//rTrig1(CLK:=xInbound);
//IF rTrig1.Q THEN
//	eState_temp1	:= '';
//	str4debug:='';
//	str4debug	:= CONCAT(STR1:=sInstanceName,STR2:='-');
//	str4debug	:= CONCAT(STR1:=str4debug,STR2:=DINT_TO_STRING(eState));
//	str4debug	:= CONCAT(STR1:=str4debug,STR2:='-');
//	str4debug	:= CONCAT(STR1:=str4debug,STR2:=strState);
//	str4debug	:= CONCAT(STR1:=str4debug,STR2:='-');
//	str4debug	:= CONCAT(STR1:=str4debug,STR2:='inbound');
//	str4debug	:= CONCAT(STR1:=str4debug,STR2:='-');
//	str4debug	:= CONCAT(STR1:=str4debug,STR2:='ON');
//	ADSLOGSTR(msgCtrlMask:=ADSLOG_MSGTYPE_LOG,msgFmtStr:=str4debug,strArg:='');
//END_IF
//fTrig1(CLK:=xInbound);
//IF eState_temp1<>strState THEN
//	eState_temp1	:= strState;
//	state_track	:= CONCAT(STR1:=state_track,STR2:=eState_temp1);
//	state_track	:= CONCAT(STR1:=state_track,STR2:='->');
//END_IF
//IF fTrig1.Q THEN
//	str4debug:='';
//	str4debug	:= CONCAT(STR1:=sInstanceName,STR2:='-');
//	str4debug	:= CONCAT(STR1:=str4debug,STR2:=DINT_TO_STRING(eState));
//	str4debug	:= CONCAT(STR1:=str4debug,STR2:='-');
//	str4debug	:= CONCAT(STR1:=str4debug,STR2:=state_track);
//	str4debug	:= CONCAT(STR1:=str4debug,STR2:='-');
//	str4debug	:= CONCAT(STR1:=str4debug,STR2:='inbound');
//	str4debug	:= CONCAT(STR1:=str4debug,STR2:='-');	
//	str4debug	:= CONCAT(STR1:=str4debug,STR2:='OFF');
//	ADSLOGSTR(msgCtrlMask:=ADSLOG_MSGTYPE_LOG,msgFmtStr:=str4debug,strArg:='');
//END_IF
IF sInstanceName='working1' THEN
	GVL.fb_autoStore1(	eModeCommand:=eModeCommand,
						eMode	=>,
						eState =>stSubModuleInfo[1].eState
					);
	stSubModuleInfo[1].Active			:= FALSE;//while on site,set to FALSE
	IF stSubModuleInfo[1].Active THEN
		eCommand:=eCommand;
	END_IF
	IF  GVL.fb_autoStore1.bUndefinedDone THEN
		bUndefinedDone := TRUE;
	END_IF	
END_IF
IF sInstanceName='working2' THEN
	GVL.fb_autoStore2(	eModeCommand:=eModeCommand,
						eMode	=>,
						eState =>stSubModuleInfo[1].eState
					);
	stSubModuleInfo[1].Active			:= FALSE;//while on site,set to FALSE
	IF stSubModuleInfo[1].Active THEN
		eCommand:=eCommand;
	END_IF	
	IF  GVL.fb_autoStore2.bUndefinedDone THEN
		bUndefinedDone := TRUE;
	END_IF		
END_IF


IF bUndefinedDone AND NOT bMachineStartedUp THEN
	eCommand	:= ePMLCommand_Abort;
	bMachineStartedUp			:= TRUE;
END_IF
//The fbStateMachine from FB_Machine gets the Information about the states and activity from the subunits
fbStateMachine.stSubUnitInfoRef.ArraySize		:= SIZEOF(stSubModuleInfo);
fbStateMachine.stSubUnitInfoRef.NoOfSubUnits	:= iSubModule;
fbStateMachine.stSubUnitInfoRef.pArray			:= ADR(stSubModuleInfo);

(*
Description: 
the callback that will be invoked when there is a publish for what the subscriber was subscribed to.
*)
METHOD Callback
VAR_INPUT
	data : PubSubData;
END_VAR

IF sInstanceName='working1' THEN
	CASE data.Topic OF	
		E_Topics.WORKING1_INBOUND_TOTE:
			IF NOT xInbound AND NOT xOutbound THEN
				xInbound	:= TRUE;
			END_IF
		E_Topics.WORKING1_OUTBOUND_TOTE:
			IF NOT xInbound AND NOT xOutbound THEN
				xOutbound	:= TRUE;
			END_IF
		E_Topics.WORKING1_BEGIN_INBOUND:
			xBeginInbound	:= TRUE;	
		E_Topics.WORKING1_ABORT_INBOUND:
			IF eStates=E_WorkingStates.WAIT_NEW_TOTE THEN
				subData.Topic	:= E_Topics.LOADING_END_OUTBOUND_WOKING1;
				GVL.PubSubService.Publish(topic:=E_Topics.LOADING_END_OUTBOUND_WOKING1,data:= subData);		
				xAbortInbound	:= TRUE;
			END_IF	
		E_Topics.WORKING1_ABORT_OUTBOUND:
			xAbortOutbound	:= TRUE;			

	END_CASE
END_IF
IF sInstanceName='working2' THEN
	CASE data.Topic OF	
		E_Topics.WORKING2_INBOUND_TOTE:
			IF NOT xInbound AND NOT xOutbound THEN
				xInbound	:= TRUE;
			END_IF
		E_Topics.WORKING2_OUTBOUND_TOTE:
			IF NOT xInbound AND NOT xOutbound THEN
				xOutbound	:= TRUE;
			END_IF
		E_Topics.WORKING2_BEGIN_INBOUND:
			xBeginInbound	:= TRUE;	
		E_Topics.WORKING2_ABORT_INBOUND:
			IF eStates=E_WorkingStates.WAIT_NEW_TOTE THEN
				subData.Topic	:= E_Topics.LOADING_END_OUTBOUND_WOKING2;
				GVL.PubSubService.Publish(topic:=E_Topics.LOADING_END_OUTBOUND_WOKING2,data:= subData);				
				xAbortInbound	:= TRUE;
			END_IF
		E_Topics.WORKING2_ABORT_OUTBOUND:
			xAbortOutbound	:= TRUE;	
		
	END_CASE
END_IF
END_METHOD

{attribute 'object_name' := 'M_Aborting'}
METHOD M_Aborting
CASE fbUnitModeManager.eModeStatus OF	
	ePMLProtUnitMode_Production, ePMLProtUnitMode_Manual:		
		roller_inbound.roller.forward			:= FALSE;
		roller_outbound.roller.forward			:= FALSE;
		roller_outbound_assist.roller.forward	:= FALSE;	
		roller_preInbound.forward				:= FALSE;
		st_mcAxis_lift.mcMoveAbsolute.Execute	:= FALSE;
		st_mcAxis_bag.mcMoveAbsolute.Execute	:= FALSE;
		st_mcAxis_lift.mcStop.Execute			:= TRUE;
		st_mcAxis_bag.mcStop.Execute			:= TRUE;	
		xInbound	:= FALSE;
		xOutbound	:= FALSE;
		bAging_test	:= FALSE;
		iAging_test	:= 0;
		CASE tote_status OF
			ToteStatus.AWAITING_INBOUND_AVAILABILITY:
			//
			ToteStatus.AWAITING_OUTBOUND_AVAILABILITY:
			//
			ToteStatus.BAG_OPEN_FAILED:
			//
			ToteStatus.DOWNSTREAM_NOT_READY:
			//
			ToteStatus.ELECTRICAL_ERROR:
			//
			ToteStatus.INBOUNDING:
			//
			ToteStatus.LOADED:
			//
			ToteStatus.MECHANICAL_ERROR:
			//
			ToteStatus.OUTBOUNDING:
			//
			ToteStatus.PERTURBING:
			//
		END_CASE
		M_StateComplete();
			
	ePMLProtUnitMode_Maintenance, ePMLUnitMode_Service:
		
		M_StateComplete();
END_CASE
END_METHOD

METHOD M_agingTest : BOOL
VAR_INPUT
	rVelocity_percent	: REAL;
END_VAR
ton_aging_test();
CASE iAging_test OF
	0://
	
	1://run forward
		ton_aging_test.PT	:= T#5S;
		ton_aging_test.IN	:= TRUE;
		st_mcAxis_lift.mcMoveAbsolute.Execute	:= TRUE;						
		st_mcAxis_lift.rActualPosSet	:= rPos_lift_up;
		st_mcAxis_lift.rVelocitySet	:= rVelocity_percent*200;
		st_mcAxis_bag.mcMoveAbsolute.Execute	:= TRUE;						
		st_mcAxis_bag.rActualPosSet	:= rPos_bag_closed;
		st_mcAxis_bag.rVelocitySet	:= rVelocity_percent*50;		
		roller_inbound.roller.forward	:= TRUE;
		roller_outbound.roller.forward	:= TRUE;
		roller_outbound_assist.roller.forward	:= TRUE;	
		roller_preInbound.forward	:= TRUE;	
		valve_lift.extend 		:= TRUE;
		valve_lift.retract		:= FALSE;
		IF st_mcAxis_lift.mcMoveAbsolute.Done AND st_mcAxis_bag.mcMoveAbsolute.Done AND ton_aging_test.Q THEN
			st_mcAxis_lift.mcMoveAbsolute.Execute	:= FALSE;
			st_mcAxis_bag.mcMoveAbsolute.Execute	:= FALSE;
			roller_inbound.roller.forward	:= FALSE;
			roller_outbound.roller.forward	:= FALSE;
			roller_outbound_assist.roller.forward	:= FALSE;	
			roller_preInbound.forward	:= FALSE;		
			ton_aging_test.IN	:= FALSE;			
			iAging_test	:= 2;
		END_IF	
	2:	
		ton_aging_test.PT	:= T#2S;
		ton_aging_test.IN	:= TRUE;
		IF ton_aging_test.Q THEN
			ton_aging_test.IN	:= FALSE;
			iAging_test	:= 3;				
		END_IF
	3://run backward
		ton_aging_test.PT	:= T#5S;
		ton_aging_test.IN	:= TRUE;
		st_mcAxis_lift.mcMoveAbsolute.Execute	:= TRUE;						
		st_mcAxis_lift.rActualPosSet	:= rPos_lift_down;
		st_mcAxis_lift.rVelocitySet	:= rVelocity_percent*200;
		st_mcAxis_bag.mcMoveAbsolute.Execute	:= TRUE;						
		st_mcAxis_bag.rActualPosSet	:= rPos_bag_opened;
		st_mcAxis_bag.rVelocitySet	:= rVelocity_percent*50;		
		roller_inbound.roller.forward	:= TRUE;
		roller_inbound.roller.backward	:= TRUE;
		roller_outbound.roller.backward	:= TRUE;
		roller_outbound_assist.roller.forward	:= TRUE;
		roller_outbound_assist.roller.backward	:= TRUE;
		roller_preInbound.forward	:= TRUE;
		roller_preInbound.backward	:= TRUE;
		valve_lift.extend 		:= FALSE;
		valve_lift.retract		:= TRUE;
		IF st_mcAxis_lift.mcMoveAbsolute.Done AND st_mcAxis_bag.mcMoveAbsolute.Done AND ton_aging_test.Q THEN
			st_mcAxis_lift.mcMoveAbsolute.Execute	:= FALSE;
			st_mcAxis_bag.mcMoveAbsolute.Execute	:= FALSE;
			roller_inbound.roller.forward	:= FALSE;
			roller_inbound.roller.backward	:= FALSE;
			roller_outbound.roller.backward	:= FALSE;
			roller_outbound_assist.roller.forward	:= FALSE;
			roller_outbound_assist.roller.backward	:= FALSE;	
			roller_preInbound.forward	:= FALSE;
			roller_preInbound.backward	:= FALSE;	
			ton_aging_test.IN	:= FALSE;			
			iAging_test	:= 4;
		END_IF	
	4:
		ton_aging_test.PT	:= T#2S;
		ton_aging_test.IN	:= TRUE;
		IF ton_aging_test.Q THEN
			diCnt_aging	:= diCnt_aging+1;
			ton_aging_test.IN	:= FALSE;
			ADSLOGSTR(msgCtrlMask:=Tc2_System.ADSLOG_MSGTYPE_LOG,msgFmtStr:=CONCAT(STR1:=sInstanceName,STR2:=DINT_TO_STRING(diCnt_aging)),strArg:='');
			iAging_test	:= 1;				
		END_IF
	
		
		
		
	10://stop
		st_mcAxis_lift.mcMoveAbsolute.Execute	:= FALSE;
		st_mcAxis_bag.mcMoveAbsolute.Execute	:= FALSE;
		roller_inbound.roller.forward	:= FALSE;
		roller_outbound.roller.forward	:= FALSE;
		roller_outbound_assist.roller.forward	:= FALSE;		
		roller_inbound.roller.backward	:= FALSE;
		roller_outbound.roller.backward	:= FALSE;
		roller_outbound_assist.roller.backward	:= FALSE;	
		roller_preInbound.forward	:= FALSE;
		roller_preInbound.backward	:= FALSE;		
		valve_lift.extend 		:= FALSE;
		valve_lift.retract		:= TRUE;
		ton_aging_test.IN	:= FALSE;	
		iAging_test	:= 0;

	END_CASE
END_METHOD

METHOD M_checkCondition : BOOL
VAR_INPUT
	condition	: E_Condition;
END_VAR

M_checkCondition	:= FALSE;
CASE condition OF
	E_Condition.NO_TOTE:
	 	IF NOT roller_inbound.photo_sensor[0].Q 
				OR NOT roller_inbound.photo_sensor[1].Q 
		THEN
			M_checkCondition	:= TRUE;
		END_IF
	E_Condition.TOTE_IN:
	 	IF  NOT roller_inbound.photo_sensor[0].Q
			AND  roller_inbound.photo_sensor[1].Q 
		THEN
			M_checkCondition	:= TRUE;
		END_IF	
	
	E_Condition.READY_LOADING_TOTE:
		//
		
	E_Condition.TOTE_READY:
		IF  ABS(AxisRef_lift.NcToPlc.ActPos-rPos_lift_down)<1 AND
			ABS(AxisRef_bag.NcToPlc.ActPos-rPos_bag_opened)<1 AND
			roller_inbound.photo_sensor[1].Q AND 
			photo_sensor_tote_detection.Q AND
			NOT roller_inbound.photo_sensor[0].Q AND 
			NOT roller_outbound.photo_sensor.Q AND
			valve_lift.retracted AND
			bagOpen_Status[0].bag_status = BagStatus.OPENED AND 
			bagOpen_Status[1].bag_status = BagStatus.OPENED 
		THEN
			tote_status	:= ToteStatus.LOADED;		
		ELSE
			IF tote_status = ToteStatus.LOADED THEN
				tote_status	:= ToteStatus.AWAITING_INBOUND_AVAILABILITY;
			END_IF
		END_IF
		
		IF NOT photo_sensor_tote_detection.Q
			AND NOT roller_inbound.photo_sensor[0].Q AND NOT roller_inbound.photo_sensor[1].Q 
			AND NOT roller_outbound.photo_sensor.Q AND valve_lift.retracted 
		THEN
			tote_status	:= ToteStatus.VACANT;	
		END_IF	
		
		IF NOT roller_inbound.photo_sensor[0].Q AND roller_inbound.photo_sensor[1].Q 
			AND photo_sensor_tote_detection.Q AND NOT roller_outbound.photo_sensor.Q 
		THEN
			IF tote_status=ToteStatus.VACANT THEN
				tote_status	:= ToteStatus.INBOUNDING;
			END_IF
		END_IF		

		M_checkCondition	:= TRUE;
END_CASE
END_METHOD

{attribute 'object_name' := 'M_Completing'}
METHOD M_Completing
CASE fbUnitModeManager.eModeStatus OF
	ePMLProtUnitMode_Production:
		;
END_CASE
END_METHOD

{attribute 'object_name' := 'M_Execute'}
METHOD M_Execute
CASE fbUnitModeManager.eModeStatus OF
	ePMLProtUnitMode_Production:		//Mode Production
		
//////////////////////////unloading///////////////////////	
				IF xOutbound THEN	
					IF M_unload() THEN
					 	xOutbound := FALSE;
					END_IF		
					RETURN;
				END_IF	
//////////////////////////loading///////////////////////
				IF xInbound THEN	
					IF M_load() THEN
						xInbound := FALSE;
					END_IF
				END_IF	

				
	ePMLProtUnitMode_Maintenance, ePMLUnitMode_Service:		
		;
	ePMLProtUnitMode_Manual:		//Manaul
	
END_CASE
END_METHOD

{attribute 'object_name' := 'M_Holding'}
METHOD M_Holding
CASE fbUnitModeManager.eModeStatus OF
	ePMLProtUnitMode_Production:		//Mode Production
		//Finisch the actual seperationstep	
		

	ePMLProtUnitMode_Maintenance:
		M_StateComplete();
END_CASE
END_METHOD

{attribute 'object_name' := 'M_Idle'}
METHOD M_Idle
ftrig_agingTest(CLK	:= bAging_test);
IF 	ftrig_agingTest.Q THEN
	iAging_test	:= 10;
END_IF
IF bAging_test THEN
	IF iAging_test=0 THEN
		iAging_test	:= 1;
	END_IF	
END_IF
M_agingTest(1.0);
END_METHOD

METHOD  M_load : BOOL
VAR_INPUT
END_VAR

VAR
	
END_VAR
M_load := FALSE;

//////////////////////////////////////////////////////////timeout//////////////////////////////////////////
		iStateTemp	:= eStateTemp;
//		ton_timeout();
		IF eStateTemp=eStates THEN
			ton_timeout.IN	:=TRUE;
		ELSE
			ton_timeout.IN	:=FALSE;
			eStateTemp	:= eStates;	
			M_Log(eLogType:=ServerityLevelType.INFO,sTextLog:='');
			IF ton_timeout.Q THEN
				RETURN;
			END_IF
		END_IF
		IF ton_timeout.Q THEN	
			ton_timeout.IN	:=FALSE;
			CASE eStates OF	
				E_LoadingStates.ERROR:	
					alarm_temp.Message	:= GenerateErrorMsg(errorType:='M',iState := iStateTemp,errorMsg:='in error state.');
				ELSE
					alarm_temp.Message	:= GenerateErrorMsg(errorType:='M',iState := iStateTemp,errorMsg:='time out');
			END_CASE
//////////////////////////////////////////////////////////states don't want to timeout and trig error//////////////////////////////////////////				
			IF  eStates<>E_WorkingStates.IDLE AND
				eStates<>E_WorkingStates.WAIT_NEW_TOTE AND
				eStates<>E_WorkingStates.WAIT AND
				eStates<>E_WorkingStates.BAG_OPEN_DETECTION AND
				eStates<>E_WorkingStates.WAIT_1 
			THEN
				tote_status	:= ToteStatus.MECHANICAL_ERROR;
				IF sInstanceName='working1' THEN					
					THIS^.pml_adminAlarm.M_SetAlarm(stAdmin:=GVL.PackTags1.Admin,stAlarm:=THIS^.alarm_temp);
				END_IF			
				IF sInstanceName='working2' THEN
					THIS^.pml_adminAlarm.M_SetAlarm(stAdmin:=GVL.PackTags2.Admin,stAlarm:=THIS^.alarm_temp);
				END_IF					
			END_IF
		END_IF
//////////////////////////////////////////////////////////conditions//////////////////////////////////////////

//////////////////////////////////////////////////////////excute//////////////////////////////////////////
CASE eStates OF 
		E_WorkingStates.IDLE:	
			st_mcAxis_lift.mcPower.Enable	:= TRUE;
			st_mcAxis_bag.mcPower.Enable	:= TRUE;
			st_mcAxis_lift.mcReset.Execute	:= TRUE;
			st_mcAxis_bag.mcReset.Execute	:= TRUE;
			tote_status	:= ToteStatus.VACANT;
			IF st_mcAxis_lift.mcReadStatus.StandStill AND st_mcAxis_bag.mcReadStatus.StandStill  THEN
				eStates	:= E_WorkingStates.INIT;
			END_IF

		E_WorkingStates.INIT:
//			ADSLOGSTR(msgCtrlMask:= ADSLOG_MSGTYPE_LOG,msgFmtStr:='load start',strArg:='');
			ton_timeout.PT	:= T#3S;		
			st_mcAxis_lift.mcMoveAbsolute.Execute	:= FALSE;
			st_mcAxis_bag.mcMoveAbsolute.Execute	:= FALSE;			
			IF M_checkCondition(condition:=E_Condition.TOTE_READY) THEN///////////avoid recieve load signal from app many times
				IF tote_status=ToteStatus.LOADED  THEN
					IF sInstanceName='working1' THEN
						eStates	:= E_WorkingStates.DONE;
					END_IF
					IF sInstanceName='working2' THEN
						eStates	:= E_WorkingStates.DONE;
					END_IF					
				ELSE
					bagOpen_Status	:= bagOpenInit_Status;					
					strLog_bagopen_detection	:= '';
					eStates	:= E_WorkingStates.BAG_OPEN_UP;
				END_IF
			END_IF		

		E_WorkingStates.BAG_OPEN_UP:	
			st_mcAxis_lift.mcMoveAbsolute.Execute	:= TRUE;		
			st_mcAxis_lift.rActualPosSet	:= rPos_lift_up;
			st_mcAxis_lift.rVelocitySet	:= 250;
			IF st_mcAxis_lift.mcMoveAbsolute.Done THEN
				st_mcAxis_lift.mcMoveAbsolute.Execute	:= FALSE;
				eStates	:= E_WorkingStates.BAG_OPEN_INIT;
			END_IF		
		E_WorkingStates.BAG_OPEN_INIT:	
			st_mcAxis_bag.mcMoveAbsolute.Execute	:= TRUE;
			st_mcAxis_bag.rVelocitySet	:= 250;
			IF bUsingOpenBag THEN
				st_mcAxis_bag.rActualPosSet	:= rPos_bag_closed;
			ELSE
				st_mcAxis_bag.rActualPosSet	:= rPos_bag_opened;
			END_IF
			IF st_mcAxis_bag.mcMoveAbsolute.Done THEN
				st_mcAxis_bag.bTouchTorque := FALSE;
				st_mcAxis_bag.mcMoveAbsolute.Execute	:= FALSE;
				eStates	:= E_WorkingStates.TOTE_LIFT_DOWN;
			END_IF				
			
		E_WorkingStates.TOTE_LIFT_DOWN:			
			valve_lift.extend	:= FALSE;
			valve_lift.retract	:= TRUE;
			IF NOT valve_lift.extended AND valve_lift.retracted THEN
				eStates	:= E_WorkingStates.WAIT_NEW_TOTE;
			END_IF	
			
//		E_WorkingStates.NOTIFY_LOADING_OUTBOUND:
//			ton_timeout.PT	:= T#1S;
//			///////////////there is no tote in working position/////////////
//			IF NOT(roller_inbound.photo_sensor[0].Q OR roller_inbound.photo_sensor[1].Q OR photo_sensor_tote_detection.Q OR roller_outbound.photo_sensor.Q) THEN
//				IF sInstanceName='working1' THEN
//					subData.Topic	:= E_Topics.LOADING_BEGIN_OUTBOUND_WOKING1;
//					GVL.PubSubService.Publish(topic:=E_Topics.LOADING_BEGIN_OUTBOUND_WOKING1,data:= subData);				
//				END_IF
//				IF sInstanceName='working2' THEN
//					subData.Topic	:= E_Topics.LOADING_BEGIN_OUTBOUND_WOKING2;
//					GVL.PubSubService.Publish(topic:=E_Topics.LOADING_BEGIN_OUTBOUND_WOKING2,data:= subData);				
//				END_IF
//				eStates	:= E_WorkingStates.WAIT_NEW_TOTE;
//			END_IF	
//			///////////////there is a tote in working position/////////////
//			IF NOT roller_inbound.photo_sensor[0].Q AND roller_inbound.photo_sensor[1].Q AND photo_sensor_tote_detection.Q AND NOT roller_outbound.photo_sensor.Q THEN
//				eStates	:= E_WorkingStates.BAG_OPEN_DOWN;
//			END_IF					
			
		E_WorkingStates.WAIT_NEW_TOTE:	
			///////////////there is a tote in working position/////////////
			IF NOT roller_inbound.photo_sensor[0].Q AND roller_inbound.photo_sensor[1].Q AND photo_sensor_tote_detection.Q AND NOT roller_outbound.photo_sensor.Q THEN
				eStates	:= E_WorkingStates.BAG_OPEN_DOWN;
			END_IF			
		/////////////////////////abort inbound command from app///////////////////
			IF xAbortInbound THEN
				xAbortInbound	:= FALSE;
				tote_status	:= ToteStatus.VACANT;
				M_load	:= TRUE;
				eStates	:= E_WorkingStates.IDLE;				
			ELSE
				tote_status	:= ToteStatus.AWAITING_INBOUND_AVAILABILITY;
			END_IF
		//////////////////////////normal process///////////////////////
			IF (xBeginInbound OR GVL.fb_loading.tote_status=ToteStatus.OUTBOUNDING) THEN
				IF sInstanceName='working1' THEN
					IF  GVL.fb_loading.valve_left_door.retracted  THEN
						xBeginInbound	:=FALSE;
						tote_status	:= ToteStatus.INBOUNDING;
						eStates	:= E_WorkingStates.WAIT_PREINBOUND_SENSOR_ON;
					END_IF					
				END_IF
				IF sInstanceName='working2' THEN
					IF GVL.fb_loading.valve_right_door.retracted THEN
						xBeginInbound	:=FALSE;
						tote_status	:= ToteStatus.INBOUNDING;
						eStates	:= E_WorkingStates.WAIT_PREINBOUND_SENSOR_ON;
					END_IF					
				END_IF
			END_IF
		/////////////////////////////while in stopping/////////////////////			
			IF  THIS^.eState = ePMLState_Stopping THEN
				IF sInstanceName='working1' THEN//publish to loading for loading might be not in stopping
					subData.Topic	:= E_Topics.LOADING_END_OUTBOUND_WOKING1;
					GVL.PubSubService.Publish(topic:=E_Topics.LOADING_END_OUTBOUND_WOKING1,data:= subData);				
				END_IF
				IF sInstanceName='working2' THEN
					subData.Topic	:= E_Topics.LOADING_END_OUTBOUND_WOKING2;
					GVL.PubSubService.Publish(topic:=E_Topics.LOADING_END_OUTBOUND_WOKING2,data:= subData);				
				END_IF
				M_load	:= TRUE;
				eStates	:= E_WorkingStates.IDLE;
			END_IF						
////////////////////////////////////////////////action/////////////////////////////////////////////
		E_WorkingStates.WAIT_PREINBOUND_SENSOR_ON:	
			ton_timeout.PT	:= T#4S;	
			roller_preInbound.forward	:= TRUE;
			IF roller_preInbound.sensor.Q THEN
				eStates	:= E_WorkingStates.WAIT_PREINBOUND_SENSOR_OFF;
			END_IF
		E_WorkingStates.WAIT_PREINBOUND_SENSOR_OFF:
			roller_preInbound.forward	:= TRUE;
			roller_inbound.roller.forward	:= TRUE;
			IF NOT roller_preInbound.sensor.Q THEN
				eStates	:= E_WorkingStates.WAIT_INBOUND_SENSOR_ON;
			END_IF		
		E_WorkingStates.WAIT_INBOUND_SENSOR_ON:	
			roller_inbound.roller.forward	:= TRUE;
			roller_preInbound.forward	:= TRUE;
			IF  roller_inbound.photo_sensor[0].Q THEN
				eStates	:= E_WorkingStates.WAIT_TOTE_DETECTION_ON;
			END_IF			
		E_WorkingStates.WAIT_TOTE_DETECTION_ON:
			roller_inbound.roller.forward	:= TRUE;
			roller_preInbound.forward	:= TRUE;
			IF photo_sensor_tote_detection.Q THEN
				eStates	:= E_WorkingStates.WAIT_INBOUND_SENSOR_OFF;
			END_IF
		E_WorkingStates.WAIT_INBOUND_SENSOR_OFF:
			roller_inbound.roller.forward	:= TRUE;
			roller_preInbound.forward	:= TRUE;
			IF NOT roller_inbound.photo_sensor[0].Q THEN
				eStates	:= E_WorkingStates.WAIT_LOAD_SENSOR_ON;
			END_IF
		E_WorkingStates.WAIT_LOAD_SENSOR_ON:
			roller_inbound.roller.forward	:= TRUE;
			roller_preInbound.forward	:= TRUE;
			IF roller_inbound.photo_sensor[1].Q THEN	
				roller_inbound.roller.forward	:= FALSE;
				roller_preInbound.forward	:= FALSE;
				eStates	:= E_WorkingStates.BAG_OPEN_DOWN;
			END_IF
		E_WorkingStates.BAG_OPEN_DOWN:
			tote_status	:= ToteStatus.INBOUNDING;
			st_mcAxis_lift.mcMoveAbsolute.Execute	:= TRUE;		
			st_mcAxis_lift.rActualPosSet	:= rPos_lift_down;
			st_mcAxis_lift.rVelocitySet	:= 250;
			IF st_mcAxis_lift.mcMoveAbsolute.Done THEN	
				eStates	:= E_WorkingStates.BAG_OPEN;
			END_IF		
		E_WorkingStates.BAG_OPEN:	
			ton_timeout.PT	:= T#3S;		
			st_mcAxis_bag.mcMoveAbsolute.Execute	:= TRUE;		
			st_mcAxis_bag.rActualPosSet	:= rPos_bag_opened;
			st_mcAxis_bag.rVelocitySet	:= 50;
			IF st_mcAxis_bag.mcMoveAbsolute.Done OR st_mcAxis_bag.bTouchTorque THEN			
				st_mcAxis_bag.mcMoveAbsolute.Execute	:= FALSE;
				eStates	:= E_WorkingStates.BAG_OPEN_DETECTION;
			END_IF	
		E_WorkingStates.BAG_OPEN_DETECTION:	
			IF ABS(st_mcAxis_bag.rActualPos-rPos_bag_opened)>5 THEN
				bagOpen_Status[0].bag_status	:= BagStatus.ERROR;
				bagOpen_Status[1].bag_status	:= BagStatus.ERROR;
				tote_status	:= ToteStatus.BAG_OPEN_FAILED;
				eStates	:= E_WorkingStates.DONE;
				RETURN;
			END_IF
			ton_timeout.PT	:= INT_TO_TIME(iDelay_sensor_detection);
			IF ton_timeout.Q THEN
				/////////////////////////////////////////////bag openner1/////////////////////////////////////////					
				FOR i:=0 TO 3 DO
					IF BagOpening_Detection[i] THEN
						bagOpen_Status[0].sensor_status	:=CONCAT(STR1:=bagOpen_Status[0].sensor_status,STR2:='1');
						bagOpen_Status[0].iCnt_sensor_detection	:=bagOpen_Status[0].iCnt_sensor_detection+1;
					ELSE
						bagOpen_Status[0].sensor_status	:=CONCAT(STR1:=bagOpen_Status[0].sensor_status,STR2:='0');
					END_IF
				END_FOR	
				IF bagOpen_Status[0].iCnt_sensor_detection>=iSensor_detection_setting[0] THEN
					bagOpen_Status[0].bag_status	:= BagStatus.OPENED;
					strLog_bagopen_detection	:= CONCAT(STR1:=bag_opening_status[0].sensor_status,STR2:='->OPENED;');
				ELSE
					bagOpen_Status[0].bag_status	:= BagStatus.ERROR;
					strLog_bagopen_detection	:= CONCAT(STR1:=bag_opening_status[0].sensor_status,STR2:='->ERROR;');
				END_IF			
				/////////////////////////////////////////////bag openner2/////////////////////////////////////////	
				FOR i:=4 TO 7 DO
					IF BagOpening_Detection[i] THEN
						bagOpen_Status[1].sensor_status	:=CONCAT(STR1:=bagOpen_Status[1].sensor_status,STR2:='1');
						bagOpen_Status[1].iCnt_sensor_detection	:=bagOpen_Status[1].iCnt_sensor_detection+1;
					ELSE
						bagOpen_Status[1].sensor_status	:=CONCAT(STR1:=bagOpen_Status[1].sensor_status,STR2:='0');
					END_IF
				END_FOR		
				IF bagOpen_Status[1].iCnt_sensor_detection>=iSensor_detection_setting[1] THEN
					bagOpen_Status[1].bag_status	:= BagStatus.OPENED;
					strLog_bagopen_detection	:= CONCAT(STR1:=bag_opening_status[1].sensor_status,STR2:='->OPENED');
				ELSE
					bagOpen_Status[1].bag_status	:= BagStatus.ERROR;
					strLog_bagopen_detection	:= CONCAT(STR1:=bag_opening_status[1].sensor_status,STR2:='->ERROR');
				END_IF				

	
				eStates	:= E_WorkingStates.TOTE_STATUS_DETECTION;	
			END_IF
		E_WorkingStates.TOTE_STATUS_DETECTION:
			IF bUsingOpenBag THEN
				IF bagOpen_Status[0].bag_status=BagStatus.OPENED AND bagOpen_Status[1].bag_status=BagStatus.OPENED THEN
					tote_status	:= ToteStatus.LOADED;
				ELSE
					tote_status	:= ToteStatus.BAG_OPEN_FAILED;
				END_IF
			ELSE
				tote_status	:= ToteStatus.LOADED;
			END_IF
			/////////////////////////////////////////writelog////////////////////////////////////////
			IF bagOpen_Status[0].bag_status=BagStatus.OPENED THEN
				strLog_bagopen_detection	:= CONCAT(STR1:=bagOpen_Status[0].sensor_status,STR2:='->OPENED;');
			ELSE	
				strLog_bagopen_detection	:= CONCAT(STR1:=bagOpen_Status[0].sensor_status,STR2:='->ERROR;');
			END_IF
			IF bagOpen_Status[1].bag_status=BagStatus.OPENED THEN
				strLog_bagopen_detection	:= CONCAT(STR1:=strLog_bagopen_detection,STR2:=bagOpen_Status[1].sensor_status);
				strLog_bagopen_detection	:= CONCAT(STR1:=strLog_bagopen_detection,STR2:='->OPENED;');
			ELSE	
				strLog_bagopen_detection	:= CONCAT(STR1:=strLog_bagopen_detection,STR2:=bagOpen_Status[1].sensor_status);
				strLog_bagopen_detection	:= CONCAT(STR1:=strLog_bagopen_detection,STR2:='->ERROR;');
			END_IF					
			eStates	:= E_WorkingStates.DONE;		
		E_WorkingStates.DONE:
			ADSLOGSTR(msgCtrlMask:= ADSLOG_MSGTYPE_LOG,msgFmtStr:=strLog_bagopen_detection,strArg:='');
			M_load	:= TRUE;
			eStates	:= E_WorkingStates.IDLE;
			

		
		
END_CASE
END_METHOD

METHOD M_mapping : BOOL
VAR_INPUT
END_VAR
IF sInstanceName='working1' THEN
	
	/////////////////////////////////////digital input-2024.5.25////////////////////////////////////////

	roller_inbound.roller.err(D:= G_IO.arDI[4].Ch[0],on_ms:=500,off_ms:=80);	
	roller_inbound.photo_sensor[0](D:= arIOLinkQualifier_Place1.CH[3].1,on_ms:=200,off_ms:=300);  //入口料框检测
	roller_inbound.photo_sensor[1](D:= arIOLinkQualifier_Place1.CH[3].0,on_ms:=100,off_ms:=100);  //X向到位感应
	
	roller_outbound.roller.err(D:= G_IO.arDI[4].Ch[1],on_ms:=500,off_ms:=80);	
	roller_outbound.photo_sensor(D:= arIOLinkQualifier_Place1.CH[4].0,on_ms:=100,off_ms:=80);   //Y向出料口感应

	roller_outbound_assist.roller.err(D:= G_IO.arDI[4].Ch[2],on_ms:=500,off_ms:=80);	
	EDM_KM            			:= G_IO.arDI[4].Ch[3];       //P24_sto反馈  
	roller_preInbound.err(D:= G_IO.arDI[4].Ch[4],on_ms:=500,off_ms:=80);	
//	roller_preInbound.sensor(D:= G_IO.arDI[4].Ch[5],on_ms:=500,off_ms:=80);	
				  
	photo_sensor_tote_detection(D:= arIOLinkQualifier_Place1.CH[4].1,on_ms:=100,off_ms:=100);  //XY对角料框感应
		
	BagOpening_Detection[0]:= arIOLinkTx_Place1[7].InputByte[1].0;
	BagOpening_Detection[1]:= arIOLinkTx_Place1[7].InputByte[0].0;
	BagOpening_Detection[2]:= arIOLinkTx_Place1[7].InputByte[1].1;
	BagOpening_Detection[3]:= arIOLinkTx_Place1[7].InputByte[0].1;
	BagOpening_Detection[4]:= arIOLinkTx_Place1[7].InputByte[1].2;
	BagOpening_Detection[5]:= arIOLinkTx_Place1[7].InputByte[0].2;
	BagOpening_Detection[6]:= arIOLinkTx_Place1[7].InputByte[1].3;
	BagOpening_Detection[7]:= arIOLinkTx_Place1[7].InputByte[0].3;
		
	valve_lift.extended		:= arIOLinkQualifier_Place1.CH[0].1 AND arIOLinkQualifier_Place1.CH[1].1;
	valve_lift.retracted	:= arIOLinkQualifier_Place1.CH[2].1 AND arIOLinkQualifier_Place1.CH[2].0;
		
	(****************************axis_lift*******************************************************)
		
	st_mcAxis_lift.limit_sensor_positive:= arIOLinkQualifier_Place1.CH[5].0	 ;
	st_mcAxis_lift.limit_sensor_negative:= arIOLinkQualifier_Place1.CH[5].1  ;
	st_mcAxis_lift.limit_sensor_home	:= arIOLinkQualifier_Place1.CH[6].1  ;
	roller_preInbound.sensor(D:= arIOLinkQualifier_Place1.CH[6].0,on_ms:=100,off_ms:=100);	
		
		
		
	(****************************axis_bagopener***************************************************)
	st_mcAxis_bag.limit_sensor_positive:= 	arIOLinkTx_Place1[7].InputByte[0].4 ;
	st_mcAxis_bag.limit_sensor_negative:= 	arIOLinkTx_Place1[7].InputByte[0].5 ;
	//using software limit position for
		
		
		
		
		
	/////////////////////////////////////digital output-2024.5.25////////////////////////////////////////
	G_IO.arDO[6].Ch[0]	:= valve_lift.extend;
	G_IO.arDO[6].Ch[1]	:= valve_lift.retract;

	G_IO.arDO[4].Ch[0]	:= roller_preInbound.forward;
	G_IO.arDO[4].Ch[1]	:= roller_preInbound.backward;		
	G_IO.arDO[4].Ch[2]	:= roller_inbound.roller.forward;
	G_IO.arDO[4].Ch[3]	:= roller_inbound.roller.backward;		
	G_IO.arDO[4].Ch[4]	:= roller_outbound.roller.backward;
	G_IO.arDO[4].Ch[5]	:= roller_outbound.roller.forward;		
	G_IO.arDO[4].Ch[6]	:= roller_outbound_assist.roller.forward;
	G_IO.arDO[4].Ch[7]	:= roller_outbound_assist.roller.backward;
			
	/////////////////////////////////////axis config////////////////////////////////////////
	mcAxis_lift
	(
		ZSN		:=   st_mcAxis_lift.limit_sensor_negative OR st_mcAxis_lift.xHoming, //TODO link to digital input
		ZSP		:=   st_mcAxis_lift.limit_sensor_positive  OR st_mcAxis_lift.xHoming, //TODO link to digital input
		IN_OUT	:= st_mcAxis_lift	, 
		AXIS	:= AxisRef_lift	, 
	);
	st_mcAxis_lift.bPosSensorShow	:= TRUE;
	st_mcAxis_lift.bNegSensorShow	:= TRUE;
	st_mcAxis_lift.bStopButtonShow	:= TRUE;
	st_mcAxis_lift.rMaxAcceleration	:= 50000;
	st_mcAxis_lift.rMaxDeceleration	:= 50000;
	st_mcAxis_lift.rMaxJerk			:= 500000;
	st_mcAxis_lift.rAcceleration	:= 2500;
	st_mcAxis_lift.rDeceleration	:= 2500;
	st_mcAxis_lift.rJerk			:= 12500;
	st_mcAxis_lift.rMaxVelocity		:= 100;
	st_mcAxis_lift.rMaxDistance		:= 50;
	st_mcAxis_lift.bPosSen	:=  st_mcAxis_lift.limit_sensor_positive ;//TODO link to digital input
	st_mcAxis_lift.bNegSen	:=  st_mcAxis_lift.limit_sensor_negative ;//TODO link to digital input
	st_mcAxis_lift.mcHome.bCalibrationCam	:= TRUE;//TODO link to digital input origin
	st_mcAxis_lift.bPositionSensor	:= TRUE;//TODO link to digital input origin
	st_mcAxis_lift.bdirFW	:= TRUE;
	st_mcAxis_lift.sNetID := '192.168.17.27.6.1';
	st_mcAxis_lift.nSlaveAddr	:= 1009;
	st_mcAxis_lift.rToqueLimitSet	:= 120;
		
	mcAxis_bag
	(
		ZSN		:=   st_mcAxis_bag.limit_sensor_negative OR st_mcAxis_bag.xHoming, //TODO link to digital input
		ZSP		:=   st_mcAxis_bag.limit_sensor_positive OR st_mcAxis_bag.xHoming, //TODO link to digital input
		IN_OUT	:= st_mcAxis_bag	, 
		AXIS	:= AxisRef_bag	, 
	);
	st_mcAxis_bag.bPosSensorShow	:= TRUE;
	st_mcAxis_bag.bNegSensorShow	:= TRUE;
	st_mcAxis_bag.bStopButtonShow	:= TRUE;
	st_mcAxis_bag.rMaxAcceleration	:= 50000;
	st_mcAxis_bag.rMaxDeceleration	:= 50000;
	st_mcAxis_bag.rMaxJerk			:= 500000;
	st_mcAxis_bag.rAcceleration	:= 500;
	st_mcAxis_bag.rDeceleration	:= 500;
	st_mcAxis_bag.rJerk			:= 2000;
	st_mcAxis_bag.rMaxVelocity		:= 300;
	st_mcAxis_bag.rMaxDistance		:= 50;
	st_mcAxis_bag.bPosSen	:=  st_mcAxis_bag.limit_sensor_positive ;//TODO link to digital input
	st_mcAxis_bag.bNegSen	:=  st_mcAxis_bag.limit_sensor_negative ;//TODO link to digital input
	st_mcAxis_bag.mcHome.bCalibrationCam	:= TRUE;//TODO link to digital input origin
	st_mcAxis_bag.bPositionSensor	:= TRUE;//TODO link to digital input origin
	st_mcAxis_bag.bdirFW	:= TRUE;
	st_mcAxis_bag.sNetID := '192.168.17.27.6.1';
	st_mcAxis_bag.nSlaveAddr	:= 1010;
	st_mcAxis_bag.rToqueLimitSet	:= 120;
	st_mcAxis_bag.rToqueSet	:= 25;
		//st_mcAxis_bag.rActTorque	:= actTorque;
//		st_mcAxis_bag.bTouque_control_enable	:=ABS(st_mcAxis_bag.rActualPos-rPos_bag_opened)>10 AND xLoading;
		
		rPos_bag_closed_step_0	:= rPos_bag_opened-rPos_bag_preopen;
END_IF
IF sInstanceName='working2' THEN
	/////////////////////////////////////digital input-2024.5.25////////////////////////////////////////

	roller_inbound.roller.err(D:= G_IO.arDI[6].Ch[0],on_ms:=500,off_ms:=80); 
	roller_inbound.photo_sensor[0](D:= arIOLinkQualifier_Place2.CH[3].1,on_ms:=100,off_ms:=80);  //入口料框检测
	roller_inbound.photo_sensor[1](D:= arIOLinkQualifier_Place2.CH[3].0,on_ms:=100,off_ms:=80);  //X向到位感应
	
	roller_outbound.roller.err(D:= G_IO.arDI[6].Ch[1],on_ms:=500,off_ms:=80); 
	roller_outbound.photo_sensor(D:= arIOLinkQualifier_Place2.CH[4].0,on_ms:=100,off_ms:=80);   //Y向出料口感应
	
	roller_outbound_assist.roller.err(D:= G_IO.arDI[6].Ch[2],on_ms:=500,off_ms:=80); 
	EDM_KM            							:= G_IO.arDI[6].Ch[3];       //P24_sto反馈  
	roller_preInbound.err(D:= G_IO.arDI[6].Ch[4],on_ms:=100,off_ms:=100);
//	roller_preInbound.sensor(D:= G_IO.arDI[6].Ch[5],on_ms:=500,off_ms:=80);	
			  
	photo_sensor_tote_detection(D:= arIOLinkQualifier_Place2.CH[4].1,on_ms:=100,off_ms:=100);  //XY对角料框感应
	
	BagOpening_Detection[0]:= arIOLinkTx_Place2[7].	InputByte[1].0;
	BagOpening_Detection[1]:= arIOLinkTx_Place2[7].	InputByte[0].0;
	BagOpening_Detection[2]:= arIOLinkTx_Place2[7].	InputByte[1].1;
	BagOpening_Detection[3]:= arIOLinkTx_Place2[7].	InputByte[0].1;
	BagOpening_Detection[4]:= arIOLinkTx_Place2[7].	InputByte[1].2;
	BagOpening_Detection[5]:= arIOLinkTx_Place2[7].	InputByte[0].2;
	BagOpening_Detection[6]:= arIOLinkTx_Place2[7].	InputByte[1].3;
	BagOpening_Detection[7]:= arIOLinkTx_Place2[7].	InputByte[0].3;
	
	
	valve_lift.extended     := arIOLinkQualifier_Place2.CH[0].1 AND arIOLinkQualifier_Place2.CH[2].1;
	valve_lift.retracted    := arIOLinkQualifier_Place2.CH[1].1 AND arIOLinkQualifier_Place2.CH[2].0;
	
	(****************************axis_lift*******************************************************)
	
	st_mcAxis_lift.limit_sensor_positive:=  arIOLinkQualifier_Place2.CH[5].0;
	st_mcAxis_lift.limit_sensor_negative:=  arIOLinkQualifier_Place2.CH[5].1;
	st_mcAxis_lift.limit_sensor_home:= 		arIOLinkQualifier_Place2.CH[6].1;
	roller_preInbound.sensor(D:= arIOLinkQualifier_Place2.CH[6].0,on_ms:=200,off_ms:=80);	
	(****************************axis_bagopener***************************************************)
	st_mcAxis_bag.limit_sensor_positive	:= arIOLinkTx_Place2[7].InputByte[0].4 ;
	st_mcAxis_bag.limit_sensor_negative	:= arIOLinkTx_Place2[7].InputByte[0].5 ;
	st_mcAxis_bag.limit_sensor_home		:= arIOLinkTx_Place2[7].InputByte[1].5 ;
	
	
	/////////////////////////////////////digital output-2024.5.25////////////////////////////////////////
	G_IO.arDO[7].Ch[0]	:= valve_lift.extend;
	G_IO.arDO[7].Ch[1]	:= valve_lift.retract;
	
	G_IO.arDO[5].Ch[0]	:= roller_preInbound.forward;
	G_IO.arDO[5].Ch[1]	:= roller_preInbound.backward;		
	G_IO.arDO[5].Ch[2]	:= roller_inbound.roller.forward;
	G_IO.arDO[5].Ch[3]	:= roller_inbound.roller.backward;	
	G_IO.arDO[5].Ch[4]	:= roller_outbound.roller.forward;
	G_IO.arDO[5].Ch[5]	:= roller_outbound.roller.backward;
	G_IO.arDO[5].Ch[6]	:= roller_outbound_assist.roller.forward;
	G_IO.arDO[5].Ch[7]	:= roller_outbound_assist.roller.backward;
	
	/////////////////////////////////////axis config////////////////////////////////////////
	mcAxis_lift
	(
		ZSN		:=   st_mcAxis_lift.limit_sensor_negative OR st_mcAxis_lift.xHoming, //TODO link to digital input
		ZSP		:=   st_mcAxis_lift.limit_sensor_positive OR st_mcAxis_lift.xHoming, //TODO link to digital input
		IN_OUT	:= st_mcAxis_lift	, 
		AXIS	:= AxisRef_lift	, 
	);
	st_mcAxis_lift.bPosSensorShow	:= TRUE;
	st_mcAxis_lift.bNegSensorShow	:= TRUE;
	st_mcAxis_lift.bStopButtonShow	:= TRUE;
	st_mcAxis_lift.rMaxAcceleration	:= 50000;
	st_mcAxis_lift.rMaxDeceleration	:= 50000;
	st_mcAxis_lift.rMaxJerk			:= 500000;
	st_mcAxis_lift.rAcceleration	:= 2500;
	st_mcAxis_lift.rDeceleration	:= 2500;
	st_mcAxis_lift.rJerk			:= 12500;
	st_mcAxis_lift.rMaxVelocity		:= 100;
	st_mcAxis_lift.rMaxDistance		:= 50;
	st_mcAxis_lift.bPosSen	:=  st_mcAxis_lift.limit_sensor_positive ;//TODO link to digital input
	st_mcAxis_lift.bNegSen	:=  st_mcAxis_lift.limit_sensor_negative ;//TODO link to digital input
	st_mcAxis_lift.mcHome.bCalibrationCam	:= TRUE;//TODO link to digital input origin
	st_mcAxis_lift.bPositionSensor	:= TRUE;//TODO link to digital input origin
	st_mcAxis_lift.bdirFW	:= TRUE;
	st_mcAxis_lift.sNetID := '192.168.17.27.7.1';
	st_mcAxis_lift.nSlaveAddr	:= 1009;
	st_mcAxis_lift.rToqueLimitSet	:= 120;
	
	mcAxis_bag
	(
		ZSN		:=   st_mcAxis_bag.limit_sensor_negative OR st_mcAxis_bag.xHoming, //TODO link to digital input
		ZSP		:=   st_mcAxis_bag.limit_sensor_positive OR st_mcAxis_bag.xHoming, //TODO link to digital input
		IN_OUT	:= st_mcAxis_bag	, 
		AXIS	:= AxisRef_bag	, 
	);
	st_mcAxis_bag.bPosSensorShow	:= TRUE;
	st_mcAxis_bag.bNegSensorShow	:= TRUE;
	st_mcAxis_bag.bStopButtonShow	:= TRUE;
	st_mcAxis_bag.rMaxAcceleration	:= 50000;
	st_mcAxis_bag.rMaxDeceleration	:= 50000;
	st_mcAxis_bag.rMaxJerk			:= 500000;
	st_mcAxis_bag.rAcceleration	:= 500;
	st_mcAxis_bag.rDeceleration	:= 500;
	st_mcAxis_bag.rJerk			:= 2000;
	st_mcAxis_bag.rMaxVelocity		:= 300;
	st_mcAxis_bag.rMaxDistance		:= 50;
	st_mcAxis_bag.bPosSen	:=  st_mcAxis_bag.limit_sensor_positive ;//TODO link to digital input
	st_mcAxis_bag.bNegSen	:=  st_mcAxis_bag.limit_sensor_negative ;//TODO link to digital input
	st_mcAxis_bag.mcHome.bCalibrationCam	:= TRUE;//TODO link to digital input origin
	st_mcAxis_bag.bPositionSensor	:= TRUE;//TODO link to digital input origin
	st_mcAxis_bag.bdirFW	:= TRUE;
	st_mcAxis_bag.sNetID := '192.168.17.27.7.1';
	st_mcAxis_bag.nSlaveAddr	:= 1010;
	st_mcAxis_bag.rToqueLimitSet	:= 120;
	st_mcAxis_bag.rToqueSet	:= 25;
	//st_mcAxis_bag.rActTorque	:= actTorque;
	//st_mcAxis_bag.bTouque_control_enable	:=ABS(st_mcAxis_bag.rActualPos-rPos_bag_opened)>10 AND xLoading;
	
	rPos_bag_closed_step_0	:= rPos_bag_opened-8;

END_IF
END_METHOD

METHOD M_Reset
VAR_INPUT
END_VAR
//Take away all commands
IF GVL.stChangeIntoProduction.bYesReset THEN
;
END_IF
END_METHOD

{attribute 'object_name' := 'M_Resetting'}
METHOD M_Resetting
CASE fbUnitModeManager.eModeStatus OF
	ePMLProtUnitMode_Production:		//Production, Mantainance, Manual
		valve_lift.extend	:= FALSE;
		valve_lift.retract	:= TRUE;
		st_mcAxis_lift.mcStop.Execute	:= FALSE;
		st_mcAxis_bag.mcStop.Execute	:= FALSE;
		st_mcAxis_lift.mcReset.Execute			:= TRUE;
		st_mcAxis_bag.mcReset.Execute			:= TRUE;		
		error_status	:= OrderToteErrorStatus.NO_ERROR;	
		ton_timeout.IN	:= FALSE;
		M_StateComplete();
	
	ePMLProtUnitMode_Maintenance, ePMLProtUnitMode_Manual, ePMLUnitMode_Service:
		M_StateComplete();
END_CASE
END_METHOD

{attribute 'object_name' := 'M_Starting'}
METHOD M_Starting
CASE fbUnitModeManager.eModeStatus OF
	ePMLProtUnitMode_Production:		//Production, Mantainance, Manual
		ton_timeout.IN	:=FALSE;
		st_mcAxis_bag.mcPower.Enable	:= TRUE;
		st_mcAxis_lift.mcPower.Enable	:= TRUE;
		IF logtech_control_command=LogTechControlCmd.TRANSFER_TOTE_FINISHED THEN		
			logtech_control_command	:= LogTechControlCmd.DO_NOTHING;	
		END_IF
		IF M_checkCondition(condition:=E_Condition.TOTE_READY) THEN
			IF tote_status = ToteStatus.LOADED OR tote_status = ToteStatus.VACANT THEN
				eStates	:= E_WorkingStates.IDLE;
				xInbound	:= FALSE;
				xOutbound	:= FALSE;
			END_IF
			IF tote_status=ToteStatus.MECHANICAL_ERROR THEN
				IF xInbound THEN
					tote_status	:= ToteStatus.INBOUNDING;
				END_IF
				IF xOutbound THEN
					tote_status	:= ToteStatus.OUTBOUNDING;
				END_IF
			END_IF			
			IF st_mcAxis_bag.mcPower.Status AND st_mcAxis_lift.mcPower.Status THEN
				M_StateComplete();
			END_IF
		END_IF
		
		
	ePMLProtUnitMode_Maintenance, ePMLProtUnitMode_Manual, ePMLUnitMode_Service:
		M_StateComplete();
END_CASE
END_METHOD

{attribute 'object_name' := 'M_Stopping'}
METHOD M_Stopping
CASE fbUnitModeManager.eModeStatus OF
	ePMLProtUnitMode_Production, ePMLProtUnitMode_Manual:
/////////////////////////////////////////////////////////	
		IF NOT xInbound AND NOT xOutbound THEN
			M_StateComplete();
			RETURN;
		END_IF
//////////////////////////unloading///////////////////////	
		IF xOutbound THEN	
			IF M_unload() THEN
			 	xOutbound := FALSE;						
				M_StateComplete();
			END_IF	
			RETURN;
		END_IF	
//////////////////////////loading///////////////////////
		IF xInbound THEN
			IF PreviousState=ePMLState_Idle THEN
				M_StateComplete();
				RETURN;	
			END_IF
				
			IF M_load() THEN
				xInbound	:= FALSE;						
				M_StateComplete();
			END_IF
		END_IF		
	

				
	ePMLProtUnitMode_Maintenance, ePMLUnitMode_Service:
		M_StateComplete();	
			//not defined
END_CASE
END_METHOD

{attribute 'object_name' := 'M_Undefined'}
METHOD M_Undefined

bUndefinedDone					:= TRUE;
END_METHOD

METHOD M_unload : BOOL
VAR_INPUT
END_VAR

M_unload := FALSE;
//event.sMethod	:= 'unload';

//////////////////////////////////////////////////////////timeout//////////////////////////////////////////
		iStateTemp	:= eStateTemp;
//		ton_timeout();
		IF eStateTemp=eStates THEN
			ton_timeout.IN	:=TRUE;
		ELSE
			ton_timeout.IN	:=FALSE;
			eStateTemp	:= eStates;	
			M_Log(eLogType:=ServerityLevelType.INFO,sTextLog:='');
			IF ton_timeout.Q THEN
				RETURN;
			END_IF
		END_IF
		IF ton_timeout.Q THEN	
			ton_timeout.IN	:=FALSE;
			CASE eStates OF	
				E_LoadingStates.ERROR:	
					alarm_temp.Message	:= GenerateErrorMsg(errorType:='M',iState := iStateTemp,errorMsg:='in error state.');
				ELSE
					alarm_temp.Message	:= GenerateErrorMsg(errorType:='M',iState := iStateTemp,errorMsg:='time out');
			END_CASE
//////////////////////////////////////////////////////////states don't want to timeout and trig error//////////////////////////////////////////				
			IF  eStates<>E_WorkingStates.IDLE AND 
				eStates<>E_WorkingStates.WAIT_UNLOADING AND 
				eStates<>E_WorkingStates.WAIT_ROBORT_IN_SAFE_PLACE AND
				eStates<>E_WorkingStates.WAIT_LOGTECH_OUTBOUND 
			THEN
				IF sInstanceName='working1' THEN
					tote_status	:= ToteStatus.MECHANICAL_ERROR;	
					THIS^.pml_adminAlarm.M_SetAlarm(stAdmin:=GVL.PackTags1.Admin,stAlarm:=THIS^.alarm_temp);					
				END_IF
				IF sInstanceName='working2' THEN
					tote_status	:= ToteStatus.MECHANICAL_ERROR;	
					THIS^.pml_adminAlarm.M_SetAlarm(stAdmin:=GVL.PackTags2.Admin,stAlarm:=THIS^.alarm_temp);					
				END_IF						

			END_IF
		END_IF
		

CASE eStates OF 
		E_WorkingStates.IDLE:
			st_mcAxis_lift.mcReset.Execute	:= TRUE;
			st_mcAxis_bag.mcReset.Execute	:= TRUE;			
			IF ton_timeout.Q THEN
				eStates	:= E_WorkingStates.INIT;
			END_IF		
		E_WorkingStates.INIT:	
			ton_timeout.PT	:= T#3S;
			bagOpen_Status	:= bagOpenInit_Status;			
			st_mcAxis_lift.mcMoveAbsolute.Execute	:= FALSE;
			st_mcAxis_bag.mcMoveAbsolute.Execute	:= FALSE;
			IF M_checkCondition(condition:=E_Condition.TOTE_READY) THEN///////////check tote status
				IF tote_status=ToteStatus.VACANT THEN
					eStates	:= E_WorkingStates.DONE;
				ELSE
					eStates	:= E_WorkingStates.WAIT_UNLOADING;
				END_IF
			END_IF		
		E_WorkingStates.WAIT_UNLOADING://wait signal from logtech and app to unload the tote
			logtech_status	:= LogTechStatus.RUNNING;//todo:remove while on site
			IF logtech_status=LogTechStatus.RUNNING THEN
				tote_status	:= ToteStatus.AWAITING_OUTBOUND_AVAILABILITY;
				IF bUsingOpenBag THEN
					eStates	:= E_WorkingStates.BAG_CLOSE_STEP_0;
				ELSE
					eStates	:= E_WorkingStates.BAG_OPEN_UP;
				END_IF				
			ELSE
				tote_status	:= ToteStatus.DOWNSTREAM_NOT_READY;
			END_IF	
		E_WorkingStates.BAG_CLOSE_STEP_0:
			IF error_status=OrderToteErrorStatus.BAG_OPEN_FAILED THEN
				st_mcAxis_bag.mcMoveAbsolute.Execute	:= TRUE;		
				st_mcAxis_bag.rActualPosSet	:= rPos_bag_closed;
				st_mcAxis_bag.rVelocitySet	:= 250;				
			ELSE
				IF NOT (ABS(st_mcAxis_bag.rActualPos-rPos_bag_closed_step_0)<0.1) THEN
					st_mcAxis_bag.mcMoveAbsolute.Execute	:= TRUE;		
					st_mcAxis_bag.rActualPosSet	:= rPos_bag_closed_step_0;
					st_mcAxis_bag.rVelocitySet	:= 250;				
				END_IF
			END_IF
			IF st_mcAxis_bag.mcMoveAbsolute.Done OR (ABS(st_mcAxis_bag.rActualPos-rPos_bag_closed_step_0)<0.1) THEN
				st_mcAxis_bag.mcMoveAbsolute.Execute	:= FALSE;
				eStates	:= E_WorkingStates.WAIT_ROBORT_IN_SAFE_PLACE;
			END_IF	
		E_WorkingStates.WAIT_ROBORT_IN_SAFE_PLACE:	
			IF bRobot_in_safety_place THEN	
				eStates	:= E_WorkingStates.BAG_OPEN_UP;
			END_IF
		E_WorkingStates.BAG_OPEN_UP:
			ton_timeout.PT	:= T#3S;
			IF bRobot_in_safety_place THEN		
				st_mcAxis_lift.mcMoveAbsolute.Execute	:= TRUE;		
				st_mcAxis_lift.rActualPosSet	:= rPos_lift_up;
				st_mcAxis_lift.rVelocitySet	:= 250;
				IF st_mcAxis_lift.mcMoveAbsolute.Done THEN
					st_mcAxis_lift.mcMoveAbsolute.Execute	:= FALSE;
					eStates	:= E_WorkingStates.TOTE_LIFT_UP;
				END_IF	
			END_IF
		E_WorkingStates.TOTE_LIFT_UP:
			valve_lift.extend	:= TRUE;
			valve_lift.retract	:= FALSE;
			IF valve_lift.extended AND NOT valve_lift.retracted THEN
				eStates	:= E_WorkingStates.WAIT_LOGTECH_OUTBOUND;
			END_IF										
		E_WorkingStates.WAIT_LOGTECH_OUTBOUND:			
			/////////////////////////abort outbound command from app///////////////////
			IF xAbortOutbound THEN
				xAbortOutbound	:= FALSE;
				tote_status	:= ToteStatus.LOADED;
				outboundTote_status	:= ToteStatus.VACANT;
				M_unload	:= TRUE;
				eStates	:= E_WorkingStates.IDLE;				
			ELSE
			//////////////////////////normal process///////////////////////
				tote_status	:= ToteStatus.AWAITING_OUTBOUND_AVAILABILITY;
				outboundTote_status	:= ToteStatus.AWAITING_INBOUND_AVAILABILITY;
				logtech_control_command	:= LogTechControlCmd.READY_TO_TRANSFER;
				logtech_transfer_status	:= LogTechTransferStatus.READY_TO_RECEIVE;//todo:remove while onsite
				IF logtech_transfer_status=LogTechTransferStatus.READY_TO_RECEIVE THEN
					eStates	:= E_WorkingStates.TOTE_UNLOAD;
				END_IF	
			END_IF			
			/////////////////////////////while in stopping/////////////////////	
			IF  eState = ePMLState_Stopping THEN
				tote_status	:= ToteStatus.LOADED;
				outboundTote_status	:= ToteStatus.VACANT;
				M_unload	:= TRUE;
				xOutbound	:= FALSE;
				eStates	:= E_WorkingStates.IDLE;
			END_IF
		E_WorkingStates.TOTE_UNLOAD:
			tote_status	:= ToteStatus.OUTBOUNDING;
			outboundTote_status	:= ToteStatus.INBOUNDING;
			logtech_control_command	:= LogTechControlCmd.TRANSFERRING_TOTE;
			valve_lift.extend	:= TRUE;
			valve_lift.retract	:= FALSE;		
			ton_timeout.PT	:= T#2S;
			roller_outbound.roller.forward		:= TRUE;
			roller_outbound_assist.roller.forward	:= TRUE;
			IF roller_outbound.photo_sensor.Q THEN
				eStates	:= E_WorkingStates.WAIT_TOTE_DETECTION_OFF;			
			END_IF	
		E_WorkingStates.WAIT_TOTE_DETECTION_OFF:	
			valve_lift.extend	:= TRUE;
			valve_lift.retract	:= FALSE;				
			roller_outbound.roller.forward		:= TRUE;
			roller_outbound_assist.roller.forward	:= TRUE;
			IF NOT photo_sensor_tote_detection.Q THEN
				eStates	:= E_WorkingStates.WAIT_SENSOR_OFF;	
			END_IF
		E_WorkingStates.WAIT_SENSOR_OFF:
			valve_lift.extend	:= TRUE;
			valve_lift.retract	:= FALSE;		
			roller_outbound.roller.forward		:= TRUE;
			roller_outbound_assist.roller.forward	:= TRUE;	
			IF NOT roller_outbound.photo_sensor.Q THEN
				eStates	:= E_WorkingStates.WAIT_RECEIVE_TOTE_FINISHED;			
			END_IF			
		E_WorkingStates.WAIT_RECEIVE_TOTE_FINISHED:
			valve_lift.extend	:= TRUE;
			valve_lift.retract	:= FALSE;			
			roller_outbound.roller.forward		:= TRUE;
			roller_outbound_assist.roller.forward	:= TRUE;
			logtech_control_command	:= LogTechControlCmd.TRANSFER_TOTE_FINISHED;
			logtech_transfer_status	:= LogTechTransferStatus.RECEIVE_TOTE_FINISHED;//todo:remove while onsite
			IF	logtech_transfer_status=LogTechTransferStatus.RECEIVE_TOTE_FINISHED THEN
				roller_outbound.roller.forward		:= FALSE;	
				roller_outbound_assist.roller.forward	:= FALSE;
				logtech_control_command	:= LogTechControlCmd.DO_NOTHING;
				eStates	:= E_WorkingStates.TOTE_LIFT_DOWN;
			END_IF
		E_WorkingStates.TOTE_LIFT_DOWN:
			roller_outbound.roller.forward		:= FALSE;	
			roller_outbound_assist.roller.forward	:= FALSE;	
			st_mcAxis_bag.mcMoveAbsolute.Execute	:= TRUE;		
			st_mcAxis_bag.rVelocitySet	:= 250;
			IF bUsingOpenBag THEN
				st_mcAxis_bag.rActualPosSet	:= rPos_bag_closed;
			ELSE
				st_mcAxis_bag.rActualPosSet	:= rPos_bag_opened;
			END_IF
			valve_lift.extend	:= FALSE;
			valve_lift.retract	:= TRUE;
			IF st_mcAxis_bag.mcMoveAbsolute.Done AND NOT valve_lift.extended AND valve_lift.retracted THEN
				st_mcAxis_bag.mcMoveAbsolute.Execute	:= FALSE;
				eStates	:= E_WorkingStates.DONE;
			END_IF				
		E_WorkingStates.DONE:	
			logtech_control_command	:= LogTechControlCmd.DO_NOTHING;
			tote_status	:= ToteStatus.VACANT;
			outboundTote_status	:= ToteStatus.LOADED;		
			M_unload	:= TRUE;
			eStates	:= E_WorkingStates.IDLE;



		
END_CASE
END_METHOD

METHOD M_waitCondition : BOOL
VAR_INPUT
	condition	: E_Condition;
END_VAR
M_waitCondition	:= FALSE;
CASE condition OF
	E_Condition.NO_TOTE:
	 	IF NOT roller_inbound.photo_sensor[1].Q THEN
			M_waitCondition	:= TRUE;
		END_IF
	E_Condition.TOTE_IN:
	 	IF roller_inbound.photo_sensor[1].Q THEN
			M_waitCondition	:= TRUE;
		END_IF	
	E_Condition.READY_LOADING_TOTE:
		IF  GVL.fb_loading.eTransfer=E_Transfer.UNLOAD
			OR tote_status=ToteStatus.LOADED 
			OR  xInbound
		THEN
			M_waitCondition	:= TRUE;
		END_IF	
END_CASE
END_METHOD

METHOD ParseStateToString : STRING
VAR_INPUT
END_VAR
CASE THIS^.eStates OF
	E_WorkingStates.IDLE:
		ParseStateToString	:='IDLE';
	E_WorkingStates.INIT:
		ParseStateToString	:='INIT';
	E_WorkingStates.CHECK:
		ParseStateToString	:='CHECK';
	E_WorkingStates.WAIT_NEW_TOTE:
		ParseStateToString	:='WAIT_NEW_TOTE';
	E_WorkingStates.LOADING:
		ParseStateToString	:='LOADING';
	E_WorkingStates.WAIT_FINISHED:
		ParseStateToString	:='WAIT_FINISHED';
	E_WorkingStates.TOTE_LOAD:
		ParseStateToString	:='TOTE_LOAD';
	E_WorkingStates.TOTE_UNLOAD:
		ParseStateToString	:='TOTE_UNLOAD';
	E_WorkingStates.BAG_OPEN:
		ParseStateToString	:='BAG_OPEN';
	E_WorkingStates.BAG_OPEN_DETECTION:
		ParseStateToString	:='BAG_OPEN_DETECTION';
	E_WorkingStates.BAG_CLOSE_STEP_0:
		ParseStateToString	:='BAG_CLOSE_STEP_0';
	E_WorkingStates.BAG_CLOSE_STEP_1:
		ParseStateToString	:='BAG_CLOSE_STEP_1';
	E_WorkingStates.BAG_CLOSE:
		ParseStateToString	:='BAG_CLOSE';
	E_WorkingStates.BAG_OPEN_INIT:
		ParseStateToString	:='BAG_OPEN_INIT';
	E_WorkingStates.TOTE_LIFT_UP:
		ParseStateToString	:='TOTE_LIFT_UP';
	E_WorkingStates.TOTE_LIFT_DOWN:
		ParseStateToString	:='TOTE_LIFT_DOWN';
	E_WorkingStates.BAG_OPEN_UP:
		ParseStateToString	:='BAG_OPEN_UP';
	E_WorkingStates.BAG_OPEN_DOWN:
		ParseStateToString	:='BAG_OPEN_DOWN';
	E_WorkingStates.TOTE_OUT:
		ParseStateToString	:='TOTE_OUT';
	E_WorkingStates.WAIT_1:
		ParseStateToString	:='WAIT_1';
	E_WorkingStates.WAIT_LOGTECH_OUTBOUND:
		ParseStateToString	:='WAIT_LOGTECH_OUTBOUND';
	E_WorkingStates.TOTE_STATUS_DETECTION:
		ParseStateToString	:='TOTE_STATUS_DETECTION';
	E_WorkingStates.NOTIFY_LOADING_OUTBOUND:
		ParseStateToString	:='NOTIFY_LOADING_OUTBOUND';
	E_WorkingStates.AGING_STATE_0:
		ParseStateToString	:='AGING_STATE_0';
	E_WorkingStates.AGING_STATE_1:
		ParseStateToString	:='AGING_STATE_1';
	E_WorkingStates.WAIT:
		ParseStateToString	:='WAIT';
	E_WorkingStates.WAIT_UNLOADING:
		ParseStateToString	:='WAIT_UNLOADING';
	E_WorkingStates.WAIT_SENSOR_ON:
		ParseStateToString	:='WAIT_SENSOR_ON';
	E_WorkingStates.WAIT_SENSOR_OFF:
		ParseStateToString	:='WAIT_SENSOR_OFF';
	E_WorkingStates.WAIT_PREINBOUND_SENSOR_ON:	
		ParseStateToString	:='WAIT_PREINBOUND_SENSOR_ON';
	E_WorkingStates.WAIT_PREINBOUND_SENSOR_OFF:	
		ParseStateToString	:='WAIT_PREINBOUND_SENSOR_OFF';		
	E_WorkingStates.WAIT_INBOUND_SENSOR_ON:
		ParseStateToString	:='WAIT_INBOUND_SENSOR_ON';
	E_WorkingStates.WAIT_INBOUND_SENSOR_OFF:
		ParseStateToString	:='WAIT_INBOUND_SENSOR_OFF';
	E_WorkingStates.WAIT_LOAD_SENSOR_ON:
		ParseStateToString	:='WAIT_LOAD_SENSOR_ON';
	E_WorkingStates.WAIT_LOAD_SENSOR_OFF:
		ParseStateToString	:='WAIT_LOAD_SENSOR_OFF';
	E_WorkingStates.WAIT_RECEIVE_TOTE_FINISHED:
		ParseStateToString	:='WAIT_RECEIVE_TOTE_FINISHED';
	E_WorkingStates.WAIT_TOTE_DETECTION_ON:
		ParseStateToString	:='WAIT_TOTE_DETECTION_ON';
	E_WorkingStates.WAIT_TOTE_DETECTION_OFF:
		ParseStateToString	:='WAIT_TOTE_DETECTION_OFF';
	E_WorkingStates.WAIT_ROBORT_IN_SAFE_PLACE:
		ParseStateToString	:='WAIT_ROBORT_IN_SAFE_PLACE';		
	E_WorkingStates.DONE:
		ParseStateToString	:='DONE';
	E_WorkingStates.ERROR:
		ParseStateToString	:='ERROR';
	ELSE
		ParseStateToString	:='UNKNOW STATE';
END_CASE
END_METHOD

END_FUNCTION_BLOCK

// ---- GlobalTextList.TcGTLO
TEXTLIST GlobalTextList
  1351 = ''
  1242 = '    UNKNOWN := 0 \n   VACANT :=  1\n      LOADED := 2\n AWAITING_INBOUND_AVAILABILITY := 3 \n      INBOUNDING := 4\n  AWAITING_OUTBOUND_AVAILABILITY:5\n    OUTBOUNDING := 6\n    PERTURBING := 7\n    UNKNOWN_ERROR := 50, \n    MECHANICAL_ERROR := 51,\n    ELECTRICAL_ERROR := 52,\n    SAFETY_ERROR := 53,\n    UPSTREAM_NOT_READY := 54,\n    TIMEOUT_WAITING_FOR_NEW_TOTE := 55,\n    DOWNSTREAM_NOT_READY := 56,\n    TIMEOUT_WAITING_FOR_SPACE := 57,\n\tBAG_OPEN_FAILED := 100'
  1602 = '    UNKNOWN := 0 \n   VACANT :=  1\n      LOADED := 2\n AWAITING_INBOUND_AVAILABILITY := 3, \n      INBOUNDING := 4,\n  AWAITING_OUTBOUND_AVAILABILITY:5, \n    OUTBOUNDING := 6,  \n    PERTURBING := 7, \n    UNKNOWN_ERROR := 50, \n    MECHANICAL_ERROR := 51,\n    ELECTRICAL_ERROR := 52,\n    SAFETY_ERROR := 53,\n    UPSTREAM_NOT_READY := 54,\n    TIMEOUT_WAITING_FOR_NEW_TOTE := 55,\n    DOWNSTREAM_NOT_READY := 56,\n    TIMEOUT_WAITING_FOR_SPACE := 57,\n\tBAG_OPEN_FAILED := 100'
  133 = '    UNKNOWN := 0 \n   VACANT :=  1\n      LOADED := 2 AWAITING_INBOUND_AVAILABILITY := 3, \n      INBOUNDING := 4,  AWAITING_OUTBOUND_AVAILABILITY:5, \n    OUTBOUNDING := 6,  \n    PERTURBING := 7, \n    UNKNOWN_ERROR := 50, \n    MECHANICAL_ERROR := 51,\n    ELECTRICAL_ERROR := 52,\n    SAFETY_ERROR := 53,\n    UPSTREAM_NOT_READY := 54,\n    TIMEOUT_WAITING_FOR_NEW_TOTE := 55,\n    DOWNSTREAM_NOT_READY := 56,\n    TIMEOUT_WAITING_FOR_SPACE := 57,\n\tBAG_OPEN_FAILED := 100'
  1738 = '    UNKNOWN := 0 \n   VACANT :=  1，\n      LOADED := 2，\n AWAITING_INBOUND_AVAILABILITY := 3, \n      INBOUNDING := 4,\n  AWAITING_OUTBOUND_AVAILABILITY:5, \n    OUTBOUNDING := 6,  \n    PERTURBING := 7, \n    UNKNOWN_ERROR := 50, \n    MECHANICAL_ERROR := 51,\n    ELECTRICAL_ERROR := 52,\n    SAFETY_ERROR := 53,\n    UPSTREAM_NOT_READY := 54,\n    TIMEOUT_WAITING_FOR_NEW_TOTE := 55,\n    DOWNSTREAM_NOT_READY := 56,\n    TIMEOUT_WAITING_FOR_SPACE := 57,\n\tBAG_OPEN_FAILED := 100'
  3042 = '    UNKNOWN := 0 \n   VACANT :=  1，\n      LOADED := 2，\n AWAITING_INBOUND_AVAILABILITY := 3, \n      INBOUNDING := 4,  AWAITING_OUTBOUND_AVAILABILITY:5, \n    OUTBOUNDING := 6,  \n    PERTURBING := 7, \n    UNKNOWN_ERROR := 50, \n    MECHANICAL_ERROR := 51,\n    ELECTRICAL_ERROR := 52,\n    SAFETY_ERROR := 53,\n    UPSTREAM_NOT_READY := 54,\n    TIMEOUT_WAITING_FOR_NEW_TOTE := 55,\n    DOWNSTREAM_NOT_READY := 56,\n    TIMEOUT_WAITING_FOR_SPACE := 57,\n\tBAG_OPEN_FAILED := 100'
  298 = '    UNKNOWN := 0 \n   VACANT :=  1，\n      LOADED := 2， AWAITING_INBOUND_AVAILABILITY := 3, \n      INBOUNDING := 4,  AWAITING_OUTBOUND_AVAILABILITY:5, \n    OUTBOUNDING := 6,  \n    PERTURBING := 7, \n    UNKNOWN_ERROR := 50, \n    MECHANICAL_ERROR := 51,\n    ELECTRICAL_ERROR := 52,\n    SAFETY_ERROR := 53,\n    UPSTREAM_NOT_READY := 54,\n    TIMEOUT_WAITING_FOR_NEW_TOTE := 55,\n    DOWNSTREAM_NOT_READY := 56,\n    TIMEOUT_WAITING_FOR_SPACE := 57,\n\tBAG_OPEN_FAILED := 100'
  387 = '    UNKNOWN := 0, \n    VACANT := 1\n    LOADED := 2,  AWAITING_INBOUND_AVAILABILITY := 3,  \n     INBOUNDING := 4,      AWAITING_OUTBOUND_AVAILABILITY := 5,  \n    OUTBOUNDING := 6,\n    PERTURBING := 7, \n    UNKNOWN_ERROR := 50, \n    MECHANICAL_ERROR := 51,\n    ELECTRICAL_ERROR := 52,\n    SAFETY_ERROR := 53,\n    UPSTREAM_NOT_READY := 54,\n    TIMEOUT_WAITING_FOR_NEW_TOTE := 55,\n    DOWNSTREAM_NOT_READY := 56,\n    TIMEOUT_WAITING_FOR_SPACE := 57,\n\t\n\tBAG_OPEN_FAILED := 100'
  1866 = '    UNKNOWN := 0, \n   VACANT :=  1,  \n      LOADED :=  2,  AWAITING_INBOUND_AVAILABILITY := 3, \n      INBOUNDING := 4,  AWAITING_OUTBOUND_AVAILABILITY:5, \n    OUTBOUNDING := 6,  \n    PERTURBING := 7, \n    UNKNOWN_ERROR := 50, \n    MECHANICAL_ERROR := 51,\n    ELECTRICAL_ERROR := 52,\n    SAFETY_ERROR := 53,\n    UPSTREAM_NOT_READY := 54,\n    TIMEOUT_WAITING_FOR_NEW_TOTE := 55,\n    DOWNSTREAM_NOT_READY := 56,\n    TIMEOUT_WAITING_FOR_SPACE := 57,\n\tBAG_OPEN_FAILED := 100'
  2213 = '    UNKNOWN := 0, \n   VACANT := 1,  \n    LOADED := 2,  AWAITING_INBOUND_AVAILABILITY := 3, \n      INBOUNDING := 4,  AWAITING_OUTBOUND_AVAILABILITY:5, \n    OUTBOUNDING := 6,  \n    PERTURBING := 7, \n    UNKNOWN_ERROR := 50, \n    MECHANICAL_ERROR := 51,\n    ELECTRICAL_ERROR := 52,\n    SAFETY_ERROR := 53,\n    UPSTREAM_NOT_READY := 54,\n    TIMEOUT_WAITING_FOR_NEW_TOTE := 55,\n    DOWNSTREAM_NOT_READY := 56,\n    TIMEOUT_WAITING_FOR_SPACE := 57,\n\tBAG_OPEN_FAILED := 100'
  972 = '    UNKNOWN := 0, \n   VACANT := 1,  \n    LOADED := 2,  AWAITING_INBOUND_AVAILABILITY := 3,  \n      INBOUNDING := 4,  AWAITING_OUTBOUND_AVAILABILITY := 5,  \n    OUTBOUNDING := 6,  \n    PERTURBING := 7, \n    UNKNOWN_ERROR := 50, \n    MECHANICAL_ERROR := 51,\n    ELECTRICAL_ERROR := 52,\n    SAFETY_ERROR := 53,\n    UPSTREAM_NOT_READY := 54,\n    TIMEOUT_WAITING_FOR_NEW_TOTE := 55,\n    DOWNSTREAM_NOT_READY := 56,\n    TIMEOUT_WAITING_FOR_SPACE := 57,\n\t\n\tBAG_OPEN_FAILED := 100'
  599 = '    UNKNOWN := 0, \n   VACANT := 1,  \n    LOADED := 2,  AWAITING_INBOUND_AVAILABILITY := 3,  \n      INBOUNDING := 4,  AWAITING_OUTBOUND_AVAILABILITY := 5,  \n    OUTBOUNDING := 6,  \n    PERTURBING := 7, \n    UNKNOWN_ERROR := 50, \n    MECHANICAL_ERROR := 51,\n    ELECTRICAL_ERROR := 52,\n    SAFETY_ERROR := 53,\n    UPSTREAM_NOT_READY := 54,\n    TIMEOUT_WAITING_FOR_NEW_TOTE := 55,\n    DOWNSTREAM_NOT_READY := 56,\n    TIMEOUT_WAITING_FOR_SPACE := 57,\n\tBAG_OPEN_FAILED := 100'
  2173 = '    UNKNOWN := 0,  (* when system is down *)\n    VACANT := 1, (* no tote here *)\n    LOADED := 2,  (* a tote loaded in current position *)\n    AWAITING_INBOUND_AVAILABILITY := 3,  (* waiting for an available inbound tote *)\n    INBOUNDING := 4,  (* inbounding tote from upper line *)\n    AWAITING_OUTBOUND_AVAILABILITY := 5,  (* waiting for an available outbound space *)\n    OUTBOUNDING := 6,  (* outbound tote to lower line *)\n    PERTURBING := 7, (* Tote vibrating *)\n\n    UNKNOWN_ERROR := 50, (* in error state, we should extend the error in the future\t*)\n    MECHANICAL_ERROR := 51,\n    ELECTRICAL_ERROR := 52,\n    SAFETY_ERROR := 53,\n    UPSTREAM_NOT_READY := 54,\n    TIMEOUT_WAITING_FOR_NEW_TOTE := 55,\n    DOWNSTREAM_NOT_READY := 56,\n    TIMEOUT_WAITING_FOR_SPACE := 57,\n\t\n\tBAG_OPEN_FAILED := 100'
  55 = ' command Products: %i'
  323 = '%.2f'
  206 = '%.2f mm'
  829 = '%.2f MPa'
  1131 = '%.2r'
  740 = '%.3f mm'
  201 = '%s'
  209 = '+'
  210 = '-'
  2384 = '2 Systems'
  54 = 'A C C I D E N T'
  18 = 'Abort'
  394 = 'ABORT INBOUND'
  2668 = 'ABORT OUTBOUND'
  33 = 'Aborted'
  34 = 'Aborting'
  602 = 'Acc'
  843 = 'Actual Position'
  830 = 'Admin'
  773 = 'Aging test'
  5 = 'Alarm'
  3043 = 'autoStore1'
  3264 = 'autoStore2'
  61 = 'Average MachSpeed: %5.2f Package/min'
  203 = 'Axis Error '
  299 = 'Axis_bagOpen_0'
  618 = 'Axis_bagOpen_1'
  211 = 'Axis_bagOpen_2'
  743 = 'Axis_bagOpen_3'
  324 = 'Axis_vacuun_0'
  786 = 'Axis_vacuun_1'
  317 = 'BAFFLE SENSOR1'
  1963 = 'BAFFLE SENSOR2'
  179 = 'BagOpen'
  63 = 'BagOpening'
  11 = 'BagOpening '
  521 = 'BagOpening-1'
  1064 = 'BagOpening_1'
  2321 = 'BagOpening_2'
  2069 = 'BagOpening_Detection'
  959 = 'Bag_)'
  1353 = 'Bag_0'
  1316 = 'Bag_1'
  1317 = 'Bag_closed'
  517 = 'Bag_opened'
  1009 = 'Bag_preopen'
  2196 = 'bDisplay'
  81 = 'BELT ESTOP'
  1803 = 'bLoad_up'
  808 = 'Breaker OFF'
  486 = 'Breaker ON'
  2216 = 'Btton Start'
  1159 = 'buffer'
  327 = 'BUFFER SAFETY'
  732 = 'Buffer Stopper'
  481 = 'bUsingOpenBag'
  1712 = 'Button stop'
  1438 = 'b_EStopRestart'
  16 = 'Clear'
  32 = 'Clearing'
  17 = 'Command'
  38 = 'Complete'
  1085 = 'Completing'
  58 = 'CurrentMachSpeed:%5.2f Package/min'
  1975 = 'DateTime'
  1723 = 'Datetime'
  349 = 'Dec'
  216 = 'deg/s'
  217 = 'deg/s²'
  50 = 'Detection\nof metal'
  180 = 'DIO'
  68 = 'Do you want to change tp production mode?'
  662 = 'DOG'
  2636 = 'DOOR CLOSED'
  2225 = 'Door Closed'
  1080 = 'Down'
  673 = 'error'
  586 = 'EStop Restart'
  2274 = 'EStopRestart'
  23 = 'Execute'
  19 = 'Execute\nComplete'
  924 = 'Extend'
  2482 = 'extend'
  614 = 'extended'
  59 = 'Finished Metalboxes: %i'
  60 = 'Finished Plasticboxes: %i'
  56 = 'Finished Products: %i '
  801 = 'Flood Light'
  1197 = 'GVL_IOLink'
  25 = 'Held'
  12 = 'Hold'
  26 = 'Holding'
  841 = 'HOME'
  248 = 'HomeDone'
  902 = 'ID'
  21 = 'Idle'
  136 = 'inbound'
  134 = 'INBOUND'
  710 = 'inbound_1'
  1624 = 'inbound_2'
  44 = 'INIT'
  4 = 'Invalid'
  1037 = 'Lamp'
  2490 = 'LIFT DOOR LEFT'
  2284 = 'LIFT DOOR RIGHT'
  668 = 'LIFT STO EDM'
  473 = 'Lift_down'
  293 = 'Lift_iuo'
  316 = 'Lift_up'
  51 = 'Light\nsensor'
  2749 = 'LIGHT STO EDM'
  319 = 'Load'
  1648 = 'Load Tote'
  1129 = 'Load Tote Request'
  762 = 'Loading'
  2693 = 'LOADING AGING'
  416 = 'Load_up'
  581 = 'Lock MCP Left Door'
  222 = 'Lock MCP Right Door'
  580 = 'Log In'
  234 = 'Log Out'
  1496 = 'LogOut'
  6 = 'Mantainance'
  7 = 'Manual'
  2290 = 'MCP ESTOP LEFT'
  1000 = 'MCP ESTOP RIGHT'
  1593 = 'MCP ESTOP2'
  708 = 'Message'
  361 = 'Method'
  2239 = 'MID SAFETY DOOR1'
  2485 = 'MID SAFETY DOOR2'
  52 = 'Move belt\n+'
  53 = 'Move to\nwork position'
  491 = 'Muanal'
  737 = 'name'
  3 = 'No'
  1516 = 'NO.'
  258 = 'NO. '
  1043 = 'None'
  1736 = 'Open MCP Left Door'
  1323 = 'Open MCP Right Door'
  711 = 'Operator'
  1406 = 'OUTBOUND'
  381 = 'outbound_1'
  1368 = 'outbound_2'
  1318 = 'outbound_assist\n\n'
  760 = 'outbound_assist_1\n\n'
  182 = 'outbound_assist_2\n\n'
  1029 = 'outbound_end'
  787 = 'Pause'
  1446 = 'photosensor'
  2037 = 'photo_sensor_bottom'
  1081 = 'photo_sensor_diagonal'
  706 = 'photo_sens[1]or_start'
  1231 = 'PICKMODULE STO EDM'
  882 = 'PICKMODULE2 STO EDM'
  1922 = 'PLACE1 STO EDM'
  1263 = 'PLACE2 STO EDM'
  1450 = 'PML '
  598 = 'Position Setting'
  1051 = 'Production'
  57 = 'Reset the Visu'
  30 = 'Reseting'
  176 = 'ROBO2T ESTOP'
  40 = 'ROBOT1 EAS'
  1399 = 'ROBOT1 EES'
  2581 = 'ROBOT1 ESTOP'
  1167 = 'ROBOT2 EAS'
  2067 = 'ROBOT2 EES'
  1126 = 'ROLLER BELT STO EDM'
  1023 = 'rolleroutbound_assist\n\n'
  1305 = 'roller_assign'
  1160 = 'roller_inbound'
  1610 = 'roller_inbound_assist'
  2157 = 'roller_outbound'
  1295 = 'roller_outbound_assist\n\n'
  2362 = 'SAFETY DOOR LEFT'
  1331 = 'SAFETYDOOR RIGHT'
  1925 = 'Sample'
  36 = 'SC'
  1012 = 'sensor[0]'
  1257 = 'sensor[1]'
  82 = 'sensor[2]'
  774 = 'sensor[3]'
  1262 = 'sensor[4]'
  1137 = 'sensor[5]'
  794 = 'sensor[6]'
  512 = 'sensor[7]'
  2929 = 'sensor_lift_atDownPos'
  681 = 'sensor_start[0]'
  1006 = 'sensor_start[1]'
  2179 = 'sensor_transfer_atFeedingPos'
  3056 = 'sensor_transfer_atWorkingPos'
  62 = 'Seperated Boxes: %i'
  415 = 'Service'
  102 = 'sStepID'
  99 = 'Jerk'
  839 = 'JOG BW'
  840 = 'JOG FW'
  1374 = 'lift'
  795 = 'LIFT'
  178 = 'Lift'
  926 = 'LIFT ESTOP'
  519 = 'LIFT STATION DETECTION'
  495 = 'LIGHT CURTAIN LEFT'
  39 = 'LIGHT CURTAIN RIGHT'
  413 = 'LOAD'
  897 = 'LOADING SAFETY'
  351 = 'Main'
  386 = 'MCP ESTOP'
  215 = 'mm/s'
  214 = 'mm/s²'
  207 = 'MOVE ABS'
  569 = 'Move relative'
  205 = 'Neg LS'
  677 = 'outbound'
  842 = 'photosensor[0]'
  79 = 'photosensor[1]'
  70 = 'photo_sensor[0]'
  919 = 'photo_sensor[1]'
  800 = 'photo_sensor_mute'
  925 = 'photo_sensor_mute_l'
  891 = 'photo_sensor_start'
  1003 = 'place'
  204 = 'Pos LS'
  844 = 'Power \nOn'
  359 = 'Power On'
  342 = 'ReM'
  1185 = 'ReM3'
  904 = 'ReM4'
  274 = 'ReM5'
  199 = 'Reset'
  10 = 'RESET'
  1651 = 'retract'
  934 = 'retracted'
  71 = 'ROBOT EAS'
  312 = 'ROBOT EES'
  72 = 'roller'
  1437 = 'Roller In'
  189 = 'roller[0]'
  709 = 'roller[1]'
  633 = 'roller[2]'
  687 = 'roller[3]'
  522 = 'roller_x'
  792 = 'roller_y'
  845 = 'RUN'
  634 = 'SAFETY DOOR'
  202 = 'SAFETY INPUT'
  617 = 'SAFETY OUTPUT'
  641 = 'sComponentID'
  438 = 'sComponent_ID'
  358 = 'sComponent_name'
  874 = 'sensor_mute'
  143 = 'sensor_mute_left'
  487 = 'sensor_mute_right'
  622 = 'Set absolute\nencoder as linear'
  454 = 'Set absolute\nencoder as rotation'
  208 = 'Set Point'
  14 = 'Set Pos to 0'
  332 = 'sEventType'
  714 = 'sEvent_MSG'
  245 = 'sID'
  220 = 'sMethod'
  1077 = 'Start'
  22 = 'Starting'
  67 = 'State Model\n%s'
  1356 = 'Station1'
  1785 = 'Station2'
  1034 = 'StepID'
  986 = 'sTime'
  198 = 'Stop'
  996 = 'STOP'
  1671 = 'stop'
  31 = 'Stopped'
  35 = 'Stopping'
  1097 = 'Suspend'
  28 = 'Suspended'
  29 = 'Suspending'
  666 = 'Time'
  2038 = 'time_detection'
  2651 = 'Tote1'
  1283 = 'Tote2'
  784 = 'tote_detection'
  3257 = 'Transfer'
  1613 = 'TryRunMode'
  590 = 'TryRunStart'
  118 = 'TryRunStop'
  585 = 'Type'
  13 = 'Unhold'
  24 = 'Unholding'
  20 = 'Unit Mode'
  780 = 'UNLOAD'
  809 = 'Unload'
  2590 = 'Unload To Left'
  297 = 'Unload To Right'
  37 = 'Unsuspend'
  27 = 'Unsuspending'
  15 = 'Unuspend'
  407 = 'UP'
  505 = 'Up'
  848 = 'User'
  8 = 'UserMode 1'
  863 = 'valve_clamp[0]'
  1846 = 'valve_left_door'
  1781 = 'valve_left_door extend'
  2324 = 'valve_left_door valve_left_door.extend'
  676 = 'valve_left_door.extend'
  1741 = 'valve_lif'
  396 = 'valve_lift'
  464 = 'valve_lift[0]'
  247 = 'valve_lift_1'
  1409 = 'valve_lift_2'
  2061 = 'valve_lif_1'
  1819 = 'valve_right_door'
  227 = 'valve_stopper'
  200 = 'Velocity'
  193 = 'WORKING SAFETY'
  246 = 'Working1'
  3242 = 'WORKING1 AGING'
  753 = 'Working1 Load'
  928 = 'Working1 Unload'
  514 = 'Working2'
  2354 = 'WORKING2 AGING'
  2337 = 'Working2 Load'
  86 = 'Working2 Unload'
  1 = 'Yes'
  2 = 'Yes, with Reset'
END_TEXTLIST

// ---- VISUs/Templates/visu_autoStore.TcVIS
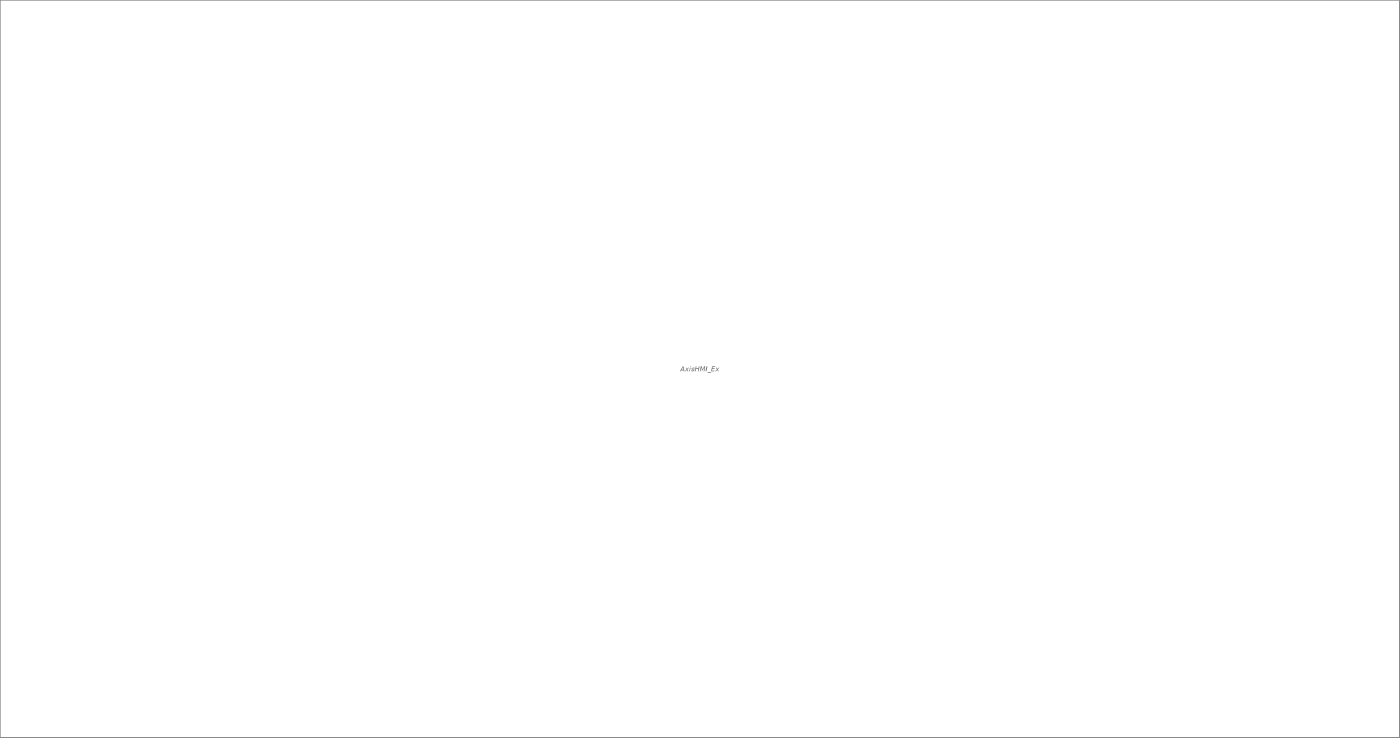
VISUALIZATION visu_autoStore  // 2048x1080
VAR_IN_OUT
	autoStore	: FB_autoStore;
END_VAR
    TabControl (0,0 2048x1080)
        shows AxisHMI_Ex(stAxisHMI := autoStore.st_mcAxis_lift, mcAxis := autoStore.mcAxis_lift, xError := autoStore.mcAxis_lift.xError)
        shows AxisHMI_Ex(stAxisHMI := autoStore.st_mcAxis_transfer, mcAxis := autoStore.mcAxis_transfer, xError := autoStore.mcAxis_transfer.xError)
        shows v_io_autoStore(autoStore := autoStore)
        shows AxisHMI_Ex(stAxisHMI := GVL.fb_working.st_mcAxis_vacuun[0], mcAxis := GVL.fb_working.mcAxis_vacuun[0], xError := GVL.fb_working.mcAxis_vacuun[0].xError)
        shows AxisHMI_Ex(stAxisHMI := GVL.fb_working.st_mcAxis_vacuun[1], mcAxis := GVL.fb_working.mcAxis_vacuun[1], xError := GVL.fb_working.mcAxis_vacuun[1].xError)
        shows AxisHMI_Ex(stAxisHMI := GVL.fb_working.st_mcAxis_bagOpen[0], mcAxis := GVL.fb_working.mcAxis_bagOpen[0], xError := GVL.fb_working.mcAxis_bagOpen[0].xError)
        shows AxisHMI_Ex(stAxisHMI := GVL.fb_working.st_mcAxis_bagOpen[1], mcAxis := GVL.fb_working.mcAxis_bagOpen[1], xError := GVL.fb_working.mcAxis_bagOpen[1].xError)
        shows AxisHMI_Ex(stAxisHMI := GVL.fb_working.st_mcAxis_bagOpen[2], mcAxis := GVL.fb_working.mcAxis_bagOpen[2], xError := GVL.fb_working.mcAxis_bagOpen[2].xError)
        shows AxisHMI_Ex(stAxisHMI := GVL.fb_working.st_mcAxis_bagOpen[3], mcAxis := GVL.fb_working.mcAxis_bagOpen[3], xError := GVL.fb_working.mcAxis_bagOpen[3].xError)
        [0]: TabTitle=Lift
        [1]: TabTitle=Transfer
        [3]: TabTitle=Axis_vacuun_0
        [4]: TabTitle=Axis_vacuun_1
        [5]: TabTitle=Axis_bagOpen_0
        [6]: TabTitle=Axis_bagOpen_1
        [7]: TabTitle=Axis_bagOpen_2
        [8]: TabTitle=Axis_bagOpen_3
        p2837713833: gantrybase.mcAxis[EN_Axis.Z].sAxisName
END_VISUALIZATION

// ---- VISUs/Templates/v_io_autoStore.TcVIS
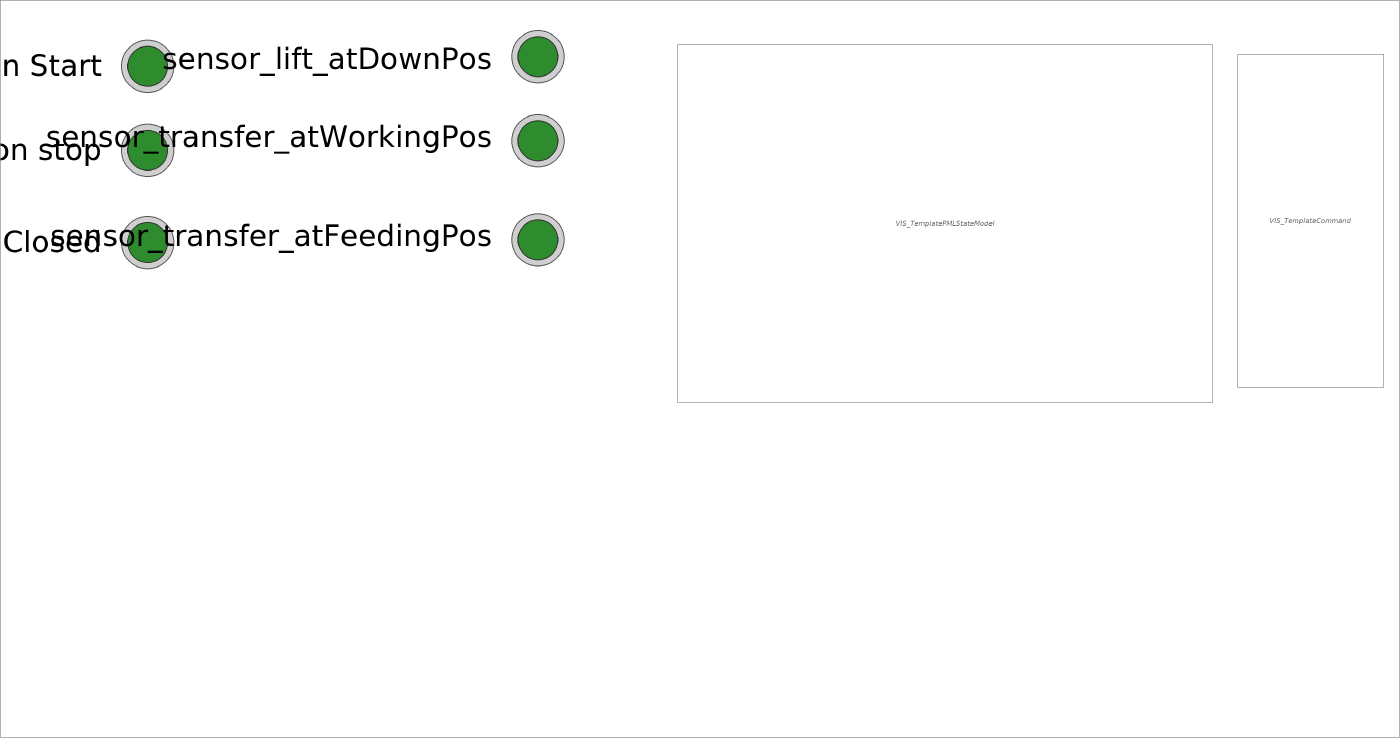
VISUALIZATION v_io_autoStore  // 2048x1080
VAR_IN_OUT
	autoStore	: FB_autoStore;
END_VAR
    Lamp1 (171,52 90x90), variable: autoStore.button_start, style: Lamp-Lamp1-Green
    Label (32,51 120x90), "Btton Start"
    Lamp1 (171,175 90x90), variable: autoStore.button_stop, style: Lamp-Lamp1-Green
    Label (32,174 120x90), "Button stop"
    Lamp1 (171,310 90x90), variable: autoStore.door_closed, style: Lamp-Lamp1-Green
    Label (32,309 120x90), "Door Closed"
    Lamp1 (742,38 90x90), variable: autoStore.sensor_lift_atDownPos, style: Lamp-Lamp1-Green
    Label (409,52 314x68), "sensor_lift_atDownPos"
    Lamp1 (742,161 90x90), variable: autoStore.sensor_transfer_atWorkingPos, style: Lamp-Lamp1-Green
    Label (339,170 384x60), "sensor_transfer_atWorkingPos"
    Lamp1 (742,306 90x90), variable: autoStore.sensor_transfer_atFeedingPos, style: Lamp-Lamp1-Green
    Label (339,315 384x60), "sensor_transfer_atFeedingPos"
    Frame (991,65 783x524)
        shows VIS_TemplatePMLStateModel(ePMLUnitMode := MAIN.fbVisu.eModeVisu, ePMLState := autoStore.eState, eStateCommand := MAIN.fbVisu.eUnitCommand)
        shows VIS_TemplatePMLStateModel()
    Frame (1810,79 214x488)
        shows VIS_TemplateCommand(eModeCommand := GVL.PackTags.Command.UnitMode, eStateCommand := autoStore.eCommand, eModeStatus := GVL.PackTags.Status.UnitModeCurrent, eStateStatus := GVL.PackTags1.Status.StateCurrent, bModeChangeReq := GVL.PackTags.Command.UnitModeChangeRequest)
END_VISUALIZATION

// ---- VISUs/VISUs/Menu.TcVIS
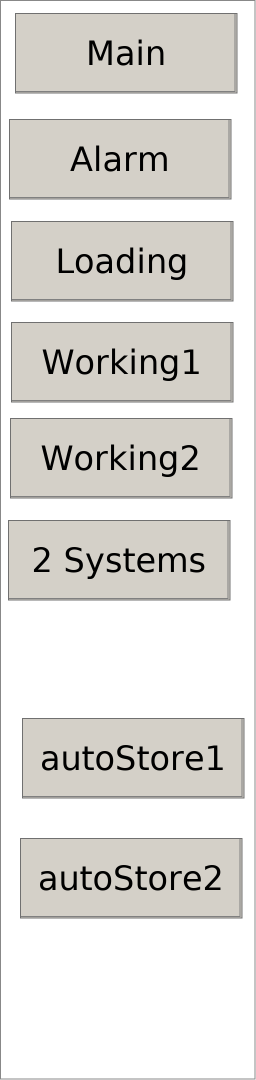
VISUALIZATION Menu  // 256x1080
    Button (9,119 222x80), "Alarm", colour toggle: G_HMI.iMainFrame =1
        p573394764: 16#FF000000 OR ( 16#FF00FF00)
        OnMouseDown: execute { G_HMI.iMainFrame	:= 1; }
    Button (15,13 222x80), "Main", colour toggle: G_HMI.iMainFrame =0
        p573394764: 16#FF000000 OR ( 16#FF00FF00)
        OnMouseDown: execute { G_HMI.iMainFrame	:= 0; }
    Button (11,221 222x80), "Loading", colour toggle: G_HMI.iMainFrame =2
        p573394764: 16#FF000000 OR ( 16#FF00FF00)
        OnMouseDown: execute { G_HMI.iMainFrame	:= 2; }
    Button (11,322 222x80), "Working1", colour toggle: G_HMI.iMainFrame =3
        p573394764: 16#FF000000 OR ( 16#FF00FF00)
        OnMouseDown: execute { G_HMI.iMainFrame	:= 3; }
    Button (10,418 222x80), "Working2", colour toggle: G_HMI.iMainFrame =4
        p573394764: 16#FF000000 OR ( 16#FF00FF00)
        OnMouseDown: execute { G_HMI.iMainFrame	:= 4; }
    Button (8,520 222x80), "2 Systems", colour toggle: G_HMI.iMainFrame =5
        p573394764: 16#FF000000 OR ( 16#FF00FF00)
        OnMouseDown: execute { G_HMI.iMainFrame	:= 5; }
    Button (22,718 222x80), "autoStore1", colour toggle: G_HMI.iMainFrame =6
        p573394764: 16#FF000000 OR ( 16#FF00FF00)
        OnMouseDown: execute { G_HMI.iMainFrame	:= 6; }
    Button (20,838 222x80), "autoStore2", colour toggle: G_HMI.iMainFrame =7
        p573394764: 16#FF000000 OR ( 16#FF00FF00)
        OnMouseDown: execute { G_HMI.iMainFrame	:= 7; }
END_VISUALIZATION

// ---- VISUs/VISUs/visu_autoStore2.TcVIS
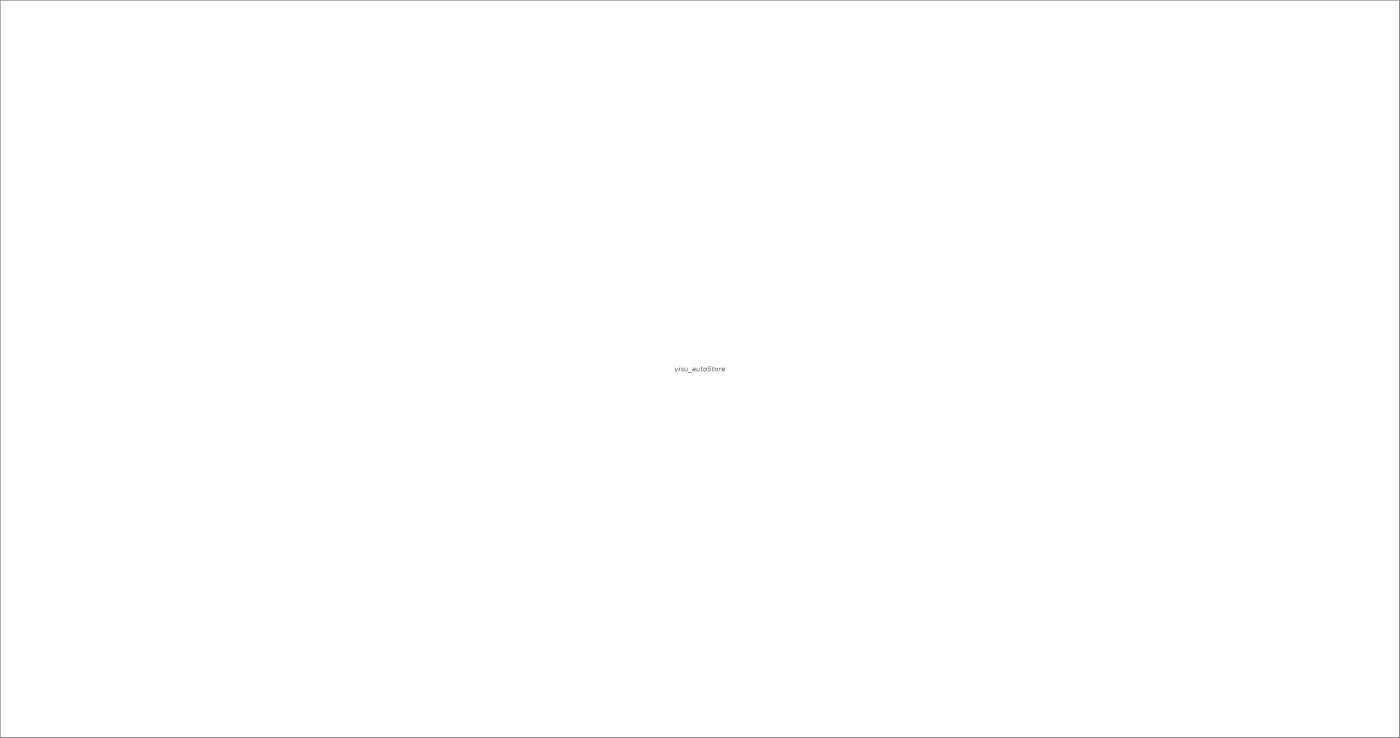
VISUALIZATION visu_autoStore2  // 2048x1080
    TabControl (0,0 2048x1080)
        shows visu_autoStore(autoStore := GVL.fb_autoStore2)
        shows AxisHMI_Ex(stAxisHMI := GVL.fb_working.st_mcAxis_vacuun[0], mcAxis := GVL.fb_working.mcAxis_vacuun[0], xError := GVL.fb_working.mcAxis_vacuun[0].xError)
        shows AxisHMI_Ex(stAxisHMI := GVL.fb_working.st_mcAxis_vacuun[1], mcAxis := GVL.fb_working.mcAxis_vacuun[1], xError := GVL.fb_working.mcAxis_vacuun[1].xError)
        shows AxisHMI_Ex(stAxisHMI := GVL.fb_working.st_mcAxis_bagOpen[0], mcAxis := GVL.fb_working.mcAxis_bagOpen[0], xError := GVL.fb_working.mcAxis_bagOpen[0].xError)
        shows AxisHMI_Ex(stAxisHMI := GVL.fb_working.st_mcAxis_bagOpen[1], mcAxis := GVL.fb_working.mcAxis_bagOpen[1], xError := GVL.fb_working.mcAxis_bagOpen[1].xError)
        shows AxisHMI_Ex(stAxisHMI := GVL.fb_working.st_mcAxis_bagOpen[2], mcAxis := GVL.fb_working.mcAxis_bagOpen[2], xError := GVL.fb_working.mcAxis_bagOpen[2].xError)
        shows AxisHMI_Ex(stAxisHMI := GVL.fb_working.st_mcAxis_bagOpen[3], mcAxis := GVL.fb_working.mcAxis_bagOpen[3], xError := GVL.fb_working.mcAxis_bagOpen[3].xError)
        shows AxisHMI_Ex(stAxisHMI := GVL.fb_working1.st_mcAxis_bag, mcAxis := GVL.fb_working1.mcAxis_bag, xError := GVL.fb_working1.mcAxis_bag.xError)
        shows v_io_working1()
        [3]: TabTitle=Axis_vacuun_0
        [4]: TabTitle=Axis_vacuun_1
        [5]: TabTitle=Axis_bagOpen_0
        [6]: TabTitle=Axis_bagOpen_1
        [7]: TabTitle=Axis_bagOpen_2
        [8]: TabTitle=Axis_bagOpen_3
        [1]: TabTitle=BagOpen
        p2837713833: gantrybase.mcAxis[EN_Axis.Z].sAxisName
END_VISUALIZATION

// ---- VISUs/VISUs/visu_operation.TcVIS
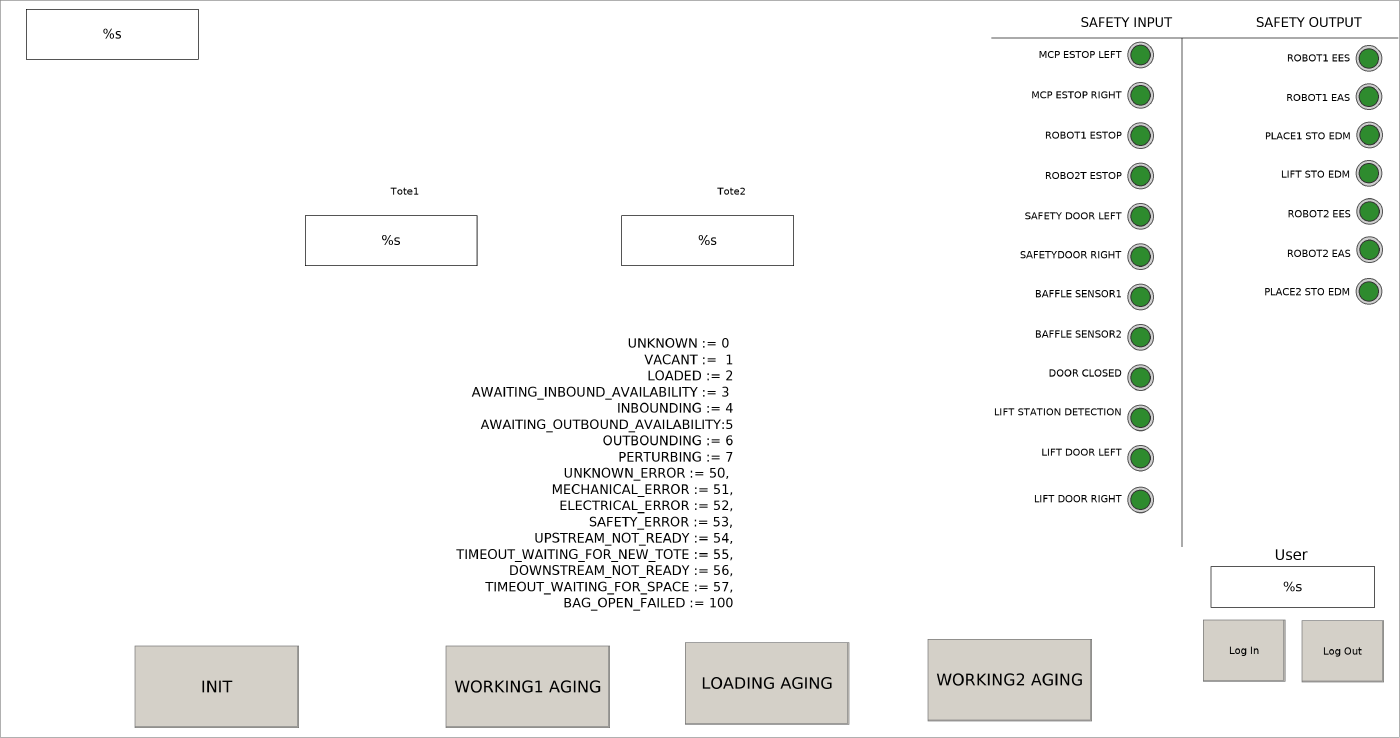
VISUALIZATION visu_operation  // 2048x1080
    Button (197,945 240x120), "INIT", colour toggle: G_HMI.bInit
        OnMouseDown: execute { G_HMI.bInit	:= TRUE; }
        OnMouseUp: execute { G_HMI.bInit	:= FALSE; }
    Lamp1 (1646,58 45x45), variable: MAIN.safety_1.mcp_estop_left.Q, style: Lamp-Lamp1-Green
    Label (1344,65 300x30), "MCP ESTOP LEFT"
    Lamp1 (1646,117 45x45), variable: MAIN.safety_1.mcp_estop_right.Q, style: Lamp-Lamp1-Green
    Label (1344,124 300x30), "MCP ESTOP RIGHT"
    Lamp1 (1646,353 45x45), variable: MAIN.safety_1.safetyDoor_right, style: Lamp-Lamp1-Green
    Label (1344,360 300x26), "SAFETYDOOR RIGHT"
    Lamp1 (1646,530 45x45), variable: MAIN.safety_1.door_closed, style: Lamp-Lamp1-Green
    Label (1344,533 300x26), "DOOR CLOSED"
    Lamp1 (1646,589 45x45), variable: MAIN.safety_1.lift_station_detection, style: Lamp-Lamp1-Green
    Label (1344,588 300x30), "LIFT STATION DETECTION"
    Lamp1 (1980,63 45x45), variable: GVL_SAFETY.robot1_STO_EES, style: Lamp-Lamp1-Green
    Label (1728,70 250x30), "ROBOT1 EES"
    Lamp1 (1980,231 45x45), variable: GVL_SAFETY.Lift_STO, style: Lamp-Lamp1-Green
    Label (1728,240 250x30), "LIFT STO EDM"
    Lamp1 (1981,175 45x45), variable: GVL_SAFETY.Place1_STO, style: Lamp-Lamp1-Green
    Label (1729,186 250x26), "PLACE1 STO EDM"
    Lamp1 (1980,404 45x45), variable: GVL_SAFETY.Place2_STO, style: Lamp-Lamp1-Green
    Label (1728,414 250x26), "PLACE2 STO EDM"
    Lamp1 (1980,119 45x45), variable: GVL_SAFETY.robot1_STO_EAS, style: Lamp-Lamp1-Green
    Label (1728,128 250x30), "ROBOT1 EAS"
    Line (1729,800) (1729,55)
    Label (1523,18 250x30), "SAFETY INPUT"
    Label (1790,18 250x30), "SAFETY OUTPUT"
    Line (1450,55) (2045,55)
    Rectangle (38,13 252x74), "%s"
    Rectangle (1771,829 240x60), "%s", text variable: G_HMI.sLoginnedUser
    Button (1904,908 120x90), "Log Out"
        OnMouseDown: VisuUserMgmt Type=Logout
    Button (1760,907 120x90), "Log In"
        OnMouseDown: VisuUserMgmt Type=Login
    Label (1814,797 150x30), "User"
    Label (1344,647 300x30), "LIFT DOOR LEFT"
    Lamp1 (1646,648 45x45), variable: MAIN.safety_1.lift_door_left.Q, style: Lamp-Lamp1-Green
    Label (1344,715 300x30), "LIFT DOOR RIGHT"
    Lamp1 (1646,709 45x45), variable: MAIN.safety_1.lift_door_right.Q, style: Lamp-Lamp1-Green
    Label (1344,301 300x30), "SAFETY DOOR LEFT"
    Lamp1 (1646,294 45x45), variable: MAIN.safety_1.safetyDoor_left, style: Lamp-Lamp1-Green
    Label (1344,415 300x30), "BAFFLE SENSOR1"
    Lamp1 (1646,412 45x45), variable: MAIN.safety_1.baffle_sensor_1, style: Lamp-Lamp1-Green
    Label (1344,474 300x30), "BAFFLE SENSOR2"
    Lamp1 (1646,471 45x45), variable: MAIN.safety_1.baffle_sensor_2, style: Lamp-Lamp1-Green
    Lamp1 (1981,287 45x45), variable: GVL_SAFETY.robot2_STO_EES, style: Lamp-Lamp1-Green
    Label (1729,298 250x30), "ROBOT2 EES"
    Lamp1 (1981,343 45x45), variable: GVL_SAFETY.robot2_STO_EAS, style: Lamp-Lamp1-Green
    Label (1729,356 250x30), "ROBOT2 EAS"
    Lamp1 (1646,176 45x45), variable: MAIN.safety_1.bRobot1_eStop, style: Lamp-Lamp1-Green
    Label (1344,183 300x30), "ROBOT1 ESTOP"
    Lamp1 (1646,235 45x45), variable: MAIN.safety_1.bRobot2_eStop, style: Lamp-Lamp1-Green
    Label (1344,242 300x30), "ROBO2T ESTOP"
    Label (316,265 300x30), "Tote1"
    Rectangle (446,315 252x74), "%s", text variable: GVL.fb_working1.tote_status
    Label (314,457 762x471), "UNKNOWN := 0 VACANT := 1 LOADED := 2 AWAITING_INBOUND_AVAILABILITY := 3 INBOUNDING := 4 AWAITING_OUTBOUND_AVAILABILITY:5 OUTBOUNDING := 6 PERTURBING := 7 UNKNOWN_ERROR := 50, MECHANICAL_ERROR := 51, ELECTRICAL_ERROR := 52, SAFETY_ERROR := 53, UPSTREAM_NOT_READY := 54, TIMEOUT_WAITING_FOR_NEW_TOTE := 55, DOWNSTREAM_NOT_READY := 56, TIMEOUT_WAITING_FOR_SPACE := 57, BAG_OPEN_FAILED := 100"
    Rectangle (909,315 252x74), "%s", text variable: GVL.fb_working2.tote_status
    Label (794,265 300x30), "Tote2"
    Button (652,945 240x120), "WORKING1 AGING"
        toggle GVL.fb_working1.bAging_test
    Button (1002,940 240x120), "LOADING AGING"
        toggle GVL.fb_loading.bAging_test
    Button (1357,935 240x120), "WORKING2 AGING"
        toggle GVL.fb_working2.bAging_test
END_VISUALIZATION

// ---- VISUs/VISUs/visu_manual.TcVIS
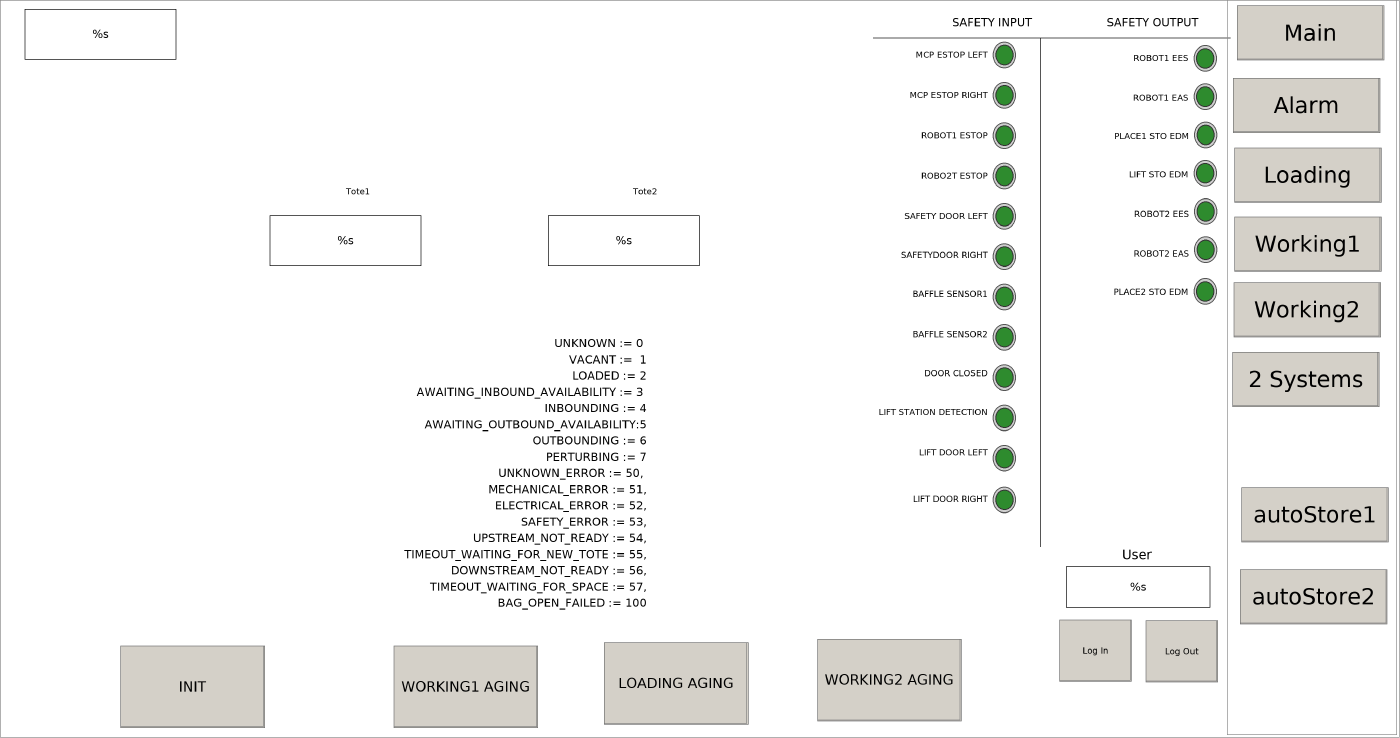
VISUALIZATION visu_manual  // 2048x1080
    Frame (3,0 1800x1080), frame switch variable: G_HMI.iMainFrame
        shows visu_operation()
        shows v_alarm()
        shows visu_loading()
        shows visu_working1()
        shows visu_working2()
        shows visu_2sys()
        shows visu_autoStore1()
        shows visu_autoStore2()
    Frame (1795,-5 248x1080), frame switch variable: G_HMI.iMainFrame
        shows Menu()
        shows visu_working()
        shows v_IO_fixtureClamp()
        shows visu_buffer()
        shows visu_loading()
        shows v_alarm()
END_VISUALIZATION

// ---- VISUs/VISUs/v_io_working2.TcVIS
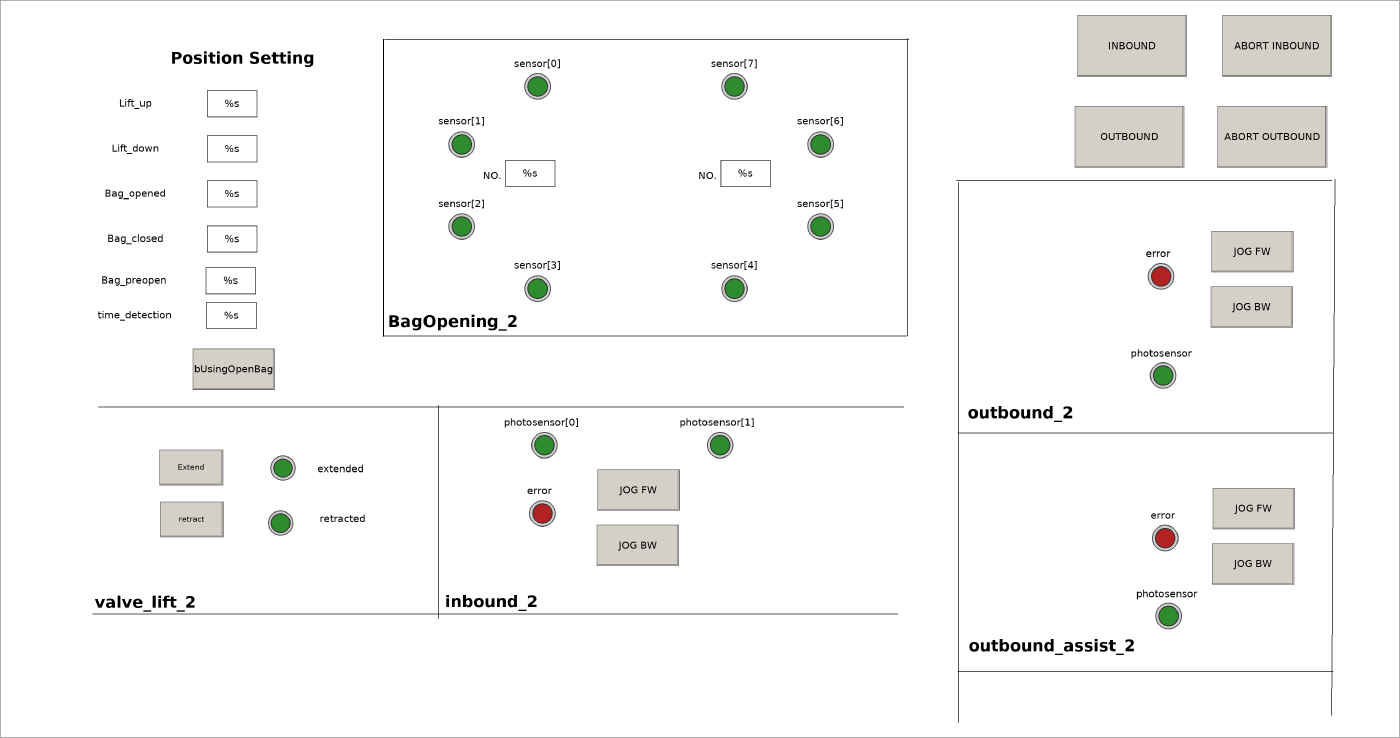
VISUALIZATION v_io_working2  // 2048x1080
    Label (91,855 244x53), "valve_lift_2"
    Button (233,658 93x52), "Extend", colour toggle: GVL.fb_working2.valve_lift.extend
        OnMouseDown: execute { GVL.fb_working2.valve_lift.extend := TRUE; GVL.fb_working2.valve_lift.retract := FALSE; }
    Button (234,734 93x52), "retract", colour toggle: GVL.fb_working2.valve_lift.retract
        OnMouseDown: execute { GVL.fb_working2.valve_lift.extend 	:= FALSE; GVL.fb_working2.valve_lift.retract 	:= TRUE; }
    Lamp1 (387,664 54x42), variable: GVL.fb_working2.valve_lift.extended, style: Lamp-Lamp1-Green
    Lamp1 (387,744 47x43), variable: GVL.fb_working2.valve_lift.retracted, style: Lamp-Lamp1-Green
    Label (432,673 132x26), "extended"
    Label (435,746 132x26), "retracted"
    Lamp1 (771,729 45x45), variable: GVL.fb_working2.roller_inbound.roller.err.Q, style: Lamp-Lamp1-Red
    Label (689,705 200x26), "error"
    Line (144,595) (1322,595)
    Button (874,687 120x60), "JOG FW", colour toggle: GVL.fb_working1.roller_inbound.roller.forward
        OnMouseDown: execute { GVL.fb_working2.roller_inbound.roller.forward	:= TRUE; }
        OnMouseUp: execute { GVL.fb_working2.roller_inbound.roller.forward	:= FALSE; }
    Button (873,768 120x60), "JOG BW", colour toggle: GVL.fb_working1.roller_inbound.roller.backward
        OnMouseDown: execute { GVL.fb_working2.roller_inbound.roller.backward	:= TRUE; }
        OnMouseUp: execute { GVL.fb_working2.roller_inbound.roller.backward	:= FALSE; }
    Lamp1 (774,629 45x45), variable: GVL.fb_working2.roller_inbound.photo_sensor[0].Q, style: Lamp-Lamp1-Green
    Label (692,605 200x26), "photosensor[0]"
    Lamp1 (1031,629 45x45), variable: GVL.fb_working2.roller_inbound.photo_sensor[1].Q, style: Lamp-Lamp1-Green
    Label (949,605 200x26), "photosensor[1]"
    Label (607,855 224x51), "inbound_2"
    Lamp1 (1676,382 45x45), variable: GVL.fb_working2.roller_outbound.roller.err.Q, style: Lamp-Lamp1-Red
    Label (1594,358 200x26), "error"
    Line (1399,264) (1948,264)
    Button (1772,338 120x60), "JOG FW", colour toggle: GVL.fb_working1.roller_outbound.roller.forward
        OnMouseDown: execute { GVL.fb_working2.roller_outbound.roller.forward	:= TRUE; }
        OnMouseUp: execute { GVL.fb_working2.roller_outbound.roller.forward	:= FALSE; }
    Button (1771,419 120x60), "JOG BW", colour toggle: GVL.fb_working1.roller_outbound.roller.backward
        OnMouseDown: execute { GVL.fb_working2.roller_outbound.roller.backward	:= TRUE; }
        OnMouseUp: execute { GVL.fb_working2.roller_outbound.roller.backward	:= FALSE; }
    Label (1375,587 236x34), "outbound_2"
    Lamp1 (1682,765 45x45), variable: GVL.fb_working2.roller_outbound_assist.roller.err.Q, style: Lamp-Lamp1-Red
    Label (1601,741 200x26), "error"
    Line (1401,633) (1950,633)
    Button (1774,714 120x60), "JOG FW", colour toggle: GVL.fb_working1.roller_outbound_assist.roller.forward
        OnMouseDown: execute { GVL.fb_working2.roller_outbound_assist.roller.forward	:= TRUE; }
        OnMouseUp: execute { GVL.fb_working2.roller_outbound_assist.roller.forward	:= FALSE; }
    Button (1773,795 120x60), "JOG BW", colour toggle: GVL.fb_working1.roller_outbound_assist.roller.backward
        OnMouseDown: execute { GVL.fb_working1.roller_outbound_assist.roller.backward	:= TRUE; }
        OnMouseUp: execute { GVL.fb_working1.roller_outbound_assist.roller.backward	:= FALSE; }
    Line (1401,982) (1950,982)
    Label (1352,940 374x68), "outbound_assist_2"
    Line (641,905) (641,593)
    Line (1948,1047) (1953,262)
    Line (1402,1057) (1402,267)
    Line (135,898) (1313,898)
    Lamp1 (764,400 45x45), variable: GVL.fb_working2.BagOpening_Detection[3], style: Lamp-Lamp1-Green
    Label (686,375 200x26), "sensor[3]"
    Lamp1 (1052,400 45x45), variable: GVL.fb_working2.BagOpening_Detection[4], style: Lamp-Lamp1-Green
    Label (974,375 200x26), "sensor[4]"
    Lamp1 (1178,309 45x45), variable: GVL.fb_working2.BagOpening_Detection[5], style: Lamp-Lamp1-Green
    Label (1100,285 200x26), "sensor[5]"
    Lamp1 (1178,189 45x45), variable: GVL.fb_working2.BagOpening_Detection[6], style: Lamp-Lamp1-Green
    Label (1100,164 200x26), "sensor[6]"
    Lamp1 (1052,104 45x45), variable: GVL.fb_working2.BagOpening_Detection[7], style: Lamp-Lamp1-Green
    Label (974,80 200x26), "sensor[7]"
    Lamp1 (764,104 45x45), variable: GVL.fb_working2.BagOpening_Detection[0], style: Lamp-Lamp1-Green
    Label (686,80 200x26), "sensor[0]"
    Lamp1 (653,189 45x45), variable: GVL.fb_working2.BagOpening_Detection[1], style: Lamp-Lamp1-Green
    Label (575,164 200x26), "sensor[1]"
    Lamp1 (653,309 45x45), variable: GVL.fb_working2.BagOpening_Detection[2], style: Lamp-Lamp1-Green
    Label (575,285 200x26), "sensor[2]"
    Line (562,57) (1329,57)
    Line (561,492) (561,57)
    Line (560,491) (1327,491)
    Line (1328,491) (1328,56)
    Rectangle (303,132 73x39), "%s", text variable: GVL.fb_working2.rPos_lift_up
        OnMouseClick: write the text variable via Default, min GVL.fb_working1.rMin_lift, max GVL.fb_working1.rMax_lift
    Rectangle (303,198 73x39), "%s", text variable: GVL.fb_working2.rPos_lift_down
        OnMouseClick: write the text variable via Default, min GVL.fb_working1.rMin_lift, max GVL.fb_working1.rMax_lift
    Rectangle (303,264 73x39), "%s", text variable: GVL.fb_working2.rPos_bag_opened
        OnMouseClick: write the text variable via Default, min GVL.fb_working1.rMin_bag, max GVL.fb_working1.rMax_bag
    Rectangle (303,330 73x39), "%s", text variable: GVL.fb_working2.rPos_bag_closed
        OnMouseClick: write the text variable via Default, min GVL.fb_working1.rMin_bag, max GVL.fb_working1.rMax_bag
    Label (98,138 200x26), "Lift_up"
    Label (98,204 200x26), "Lift_down"
    Label (98,270 200x26), "Bag_opened"
    Label (98,336 200x26), "Bag_closed"
    Label (180,72 350x26), "Position Setting"
    Rectangle (739,234 73x39), "%s", text variable: GVL.fb_working2.iSensor_detection_setting[0]
        OnMouseClick: write the text variable via Default, min 3, max 4
    Label (670,244 100x26), "NO."
    Rectangle (1054,234 73x39), "%s", text variable: GVL.fb_working2.iSensor_detection_setting[1]
        OnMouseClick: write the text variable via Default, min 3, max 4
    Label (985,244 100x26), "NO."
    Label (447,416 432x109), "BagOpening_2"
    Lamp1 (1679,527 45x45), variable: GVL.fb_working2.photo_sensor_tote_detection.Q, style: Lamp-Lamp1-Green
    Label (1599,504 200x26), "photosensor"
    Lamp1 (1687,879 45x45), variable: GVL.fb_working2.roller_outbound.photo_sensor.Q, style: Lamp-Lamp1-Green
    Label (1607,856 200x26), "photosensor"
    Rectangle (301,391 73x39), "%s", text variable: GVL.fb_working2.rPos_bag_preopen
        OnMouseClick: write the text variable via Default, min GVL.fb_working2.rMin_bag, max 15
    Label (96,397 200x26), "Bag_preopen"
    Rectangle (302,442 73x39), "%s", text variable: GVL.fb_working2.iDelay_sensor_detection
        OnMouseClick: write the text variable via Default, min 100, max 500
    Label (97,448 200x26), "time_detection"
    Button (1576,22 160x90), "INBOUND", colour toggle: MAIN.tote_2.bInbound
        OnMouseUp: execute { MAIN.tote_2.bInbound	:= TRUE; }
    Button (1572,155 160x90), "OUTBOUND", colour toggle: MAIN.tote_2.bOutbound
        OnMouseUp: execute { MAIN.tote_2.bOutbound	:= TRUE; }
    Button (1788,22 160x90), "ABORT INBOUND", colour toggle: MAIN.tote_2.bAbortInbound
        OnMouseUp: execute { MAIN.tote_2.bAbortInbound	:= TRUE; }
    Button (1781,155 160x90), "ABORT OUTBOUND", colour toggle: MAIN.tote_2.bAbortOutbound
        OnMouseUp: execute { MAIN.tote_2.bAbortOutbound	:= TRUE; }
    Button (282,510 120x60), "bUsingOpenBag", colour toggle: GVL.fb_working2.bUsingOpenBag
        toggle GVL.fb_working2.bUsingOpenBag
END_VISUALIZATION
